(* PLC project Система умного дома.project, CODESYS CODESYS V3.5 SP17 Patch 3 *)
(* stored: creationDateTime 2026-04-06T20:38:17.5908527, modificationDateTime 2026-03-25T09:46:39.3897592 *)

TYPE E_ALERT_PRIORITY : (ALERT_PRIORITY_NONE := 0, ALERT_PRIORITY_LOW := 1, ALERT_PRIORITY_MEDIUM := 2, ALERT_PRIORITY_HIGH := 3, ALERT_PRIORITY_CRITICAL := 4) USINT;
END_TYPE

TYPE E_Adapt_Profile : (ADAPT_PROFILE_STABLE := 0, ADAPT_PROFILE_BALANCED := 1, ADAPT_PROFILE_AGGRESSIVE := 2) USINT;
END_TYPE

TYPE E_Behavior_Mode : (BEHAVIOR_HOME := 0, BEHAVIOR_AWAY := 1, BEHAVIOR_NIGHT := 2, BEHAVIOR_MAINTENANCE := 3) INT;
END_TYPE

TYPE E_FABRIC_LIFECYCLE_STATE : (FABRIC_INITIALIZING := 0, FABRIC_ACTIVE := 1, FABRIC_DEGRADED := 2, FABRIC_PASSIVE := 3, FABRIC_QUARANTINED := 4, FABRIC_SUSPENDED := 5) INT;
END_TYPE

TYPE E_GOVERNANCE_PRIORITY_TIER : (TIER_0_SAFETY := 0, TIER_1_AUTHORITY := 1, TIER_2_PHYSICAL_TRUTH := 2, TIER_3_SURVIVABILITY := 3, TIER_4_OBSERVABILITY := 4, TIER_5_ANALYTICS := 5) INT;
END_TYPE

TYPE E_Gateway_Command_Type : (CMD_NONE := 0, CMD_SET_SCENARIO := 1, CMD_SET_LIGHT := 2, CMD_SET_SOCKET := 3, CMD_SET_SECURITY := 4, CMD_SET_TEMP := 5, CMD_SET_VENT := 6, CMD_SET_BLINDS := 7, CMD_TELEGRAM_MSG := 8, CMD_SYNC_TIME := 9, CMD_RESET_ERRORS := 10, CMD_SET_CONFIG := 11) USINT;
END_TYPE

TYPE E_Heating_Allocation_Block_Reason : (NONE := 0, PRESSURE_UNAVAILABLE := 1, SERVICE_DISABLED := 2, PREDICTIVE_DEGRADED := 3, POLICY_BUDGET_SHED := 4, FREEZE_BYPASS := 5, DHW_BYPASS := 6) INT;
END_TYPE

TYPE E_Heating_Policy_Mode : (HPM_NORMAL := 0, HPM_DEGRADED := 1, HPM_FREEZE_PROTECT := 2, HPM_MAINTENANCE := 3, HPM_SAFETY_BLOCK := 4, HPM_FAULT_ISOLATION := 5) INT;
END_TYPE

TYPE E_Heating_RootCause : (RC_NONE := 0, RC_EMERGENCY_STOP := 1, RC_GAS_SAFETY := 2, RC_IO_OFFLINE := 3, RC_BOILER_OFFLINE := 4, RC_BOILER_ERROR := 5, RC_NO_FLAME := 6, RC_NO_FLOW := 7, RC_PUMP_FAILURE := 8, RC_VALVES_CLOSED := 9, RC_NO_HEAT_TRANSFER := 10, RC_LOW_SUPPLY_TEMP := 11, RC_SENSOR_ERROR := 12, RC_POLICY_BLOCKED := 13, RC_UNKNOWN := 14) INT;
END_TYPE

TYPE E_Heating_Runtime_Phase : (HRP_DISABLED := 0, HRP_IDLE := 10, HRP_DHW := 20, HRP_HEATING := 30, HRP_SERVICE_GATING := 40, HRP_STATE_PUBLICATION := 50, HRP_DIAGNOSTICS := 60, HRP_OUTPUT_PROJECTION := 70, HRP_COMPLETE := 100, HRP_FAULT := 900) INT;
END_TYPE

TYPE E_Lifetime_Device_Type : (LIFETIME_DEVICE_PUMP := 1, LIFETIME_DEVICE_FAN := 2) USINT;
END_TYPE

TYPE E_Modbus_Function : (MB_NONE := 0, MB_FC03_READ_HOLDING_REGISTERS := 3, MB_FC04_READ_INPUT_REGISTERS := 4, MB_FC06_WRITE_SINGLE_REGISTER := 6, MB_FC16_WRITE_MULTIPLE_REGISTERS := 16) INT;
END_TYPE

TYPE E_Modbus_RTU_RX_State : (MB_RTU_RX_IDLE := 0, MB_RTU_RX_RECEIVING := 1, MB_RTU_RX_FRAME_READY := 2, MB_RTU_RX_CRC_ERROR := 3, MB_RTU_RX_OVERFLOW := 4, MB_RTU_RX_SHORT_FRAME := 5) INT;
END_TYPE

TYPE E_Modbus_SysCom_Backend_State : (MB_SYSCOM_CLOSED := 0, MB_SYSCOM_OPENING := 1, MB_SYSCOM_ONLINE := 2, MB_SYSCOM_ERROR := 3, MB_SYSCOM_RECONNECT_WAIT := 4) INT;
END_TYPE

TYPE E_OpenTherm_Adapter_State : (OT_STATE_OFFLINE := 0, OT_STATE_ONLINE := 1, OT_STATE_HEARTBEAT_TIMEOUT := 2, OT_STATE_ACK_TIMEOUT := 3, OT_STATE_ADAPTER_ERROR := 4) INT;
END_TYPE

TYPE E_OpenTherm_Error : (OT_ERROR_NONE := 0, OT_ERROR_HEARTBEAT_TIMEOUT := 1, OT_ERROR_ACK_TIMEOUT := 2, OT_ERROR_ADAPTER_FAULT := 3, OT_ERROR_COMMUNICATION := 4, OT_ERROR_INVALID_RESPONSE := 5) INT;
END_TYPE

TYPE E_Outdoor_Mode : (OUTDOOR_MODE_AUTO := 0, OUTDOOR_MODE_PARTY := 1, OUTDOOR_MODE_SECURITY := 2, OUTDOOR_MODE_ECONOMY := 3, OUTDOOR_MODE_MANUAL := 4) USINT;
END_TYPE

TYPE E_PLC_ROLE : (ROLE_UNDEFINED := 0, ROLE_ACTIVE := 1, ROLE_STANDBY := 2, ROLE_OFFLINE := 3) USINT;
END_TYPE

TYPE E_RUNTIME_ADAPTIVE_MODE : (FULL_SEMANTIC_MODE := 0, REDUCED_ANALYTICS_MODE := 1, SURVIVABILITY_MODE := 2, MINIMAL_SAFE_MODE := 3) INT;
END_TYPE

TYPE E_RUNTIME_TRANSITION_RESULT : (TRANSITION_VALID := 0, TRANSITION_FORBIDDEN := 1, TRANSITION_REQUIRES_PROOF := 2, TRANSITION_REQUIRES_RECOVERY := 3, TRANSITION_REQUIRES_TEMPORAL_ALIGNMENT := 4) INT;
END_TYPE

TYPE E_Recovery_Phase : (IDLE := 0, STABILIZING := 1, WAIT_MANUAL_CONFIRM := 2, RECOVERING := 3, COOLDOWN := 4, ABORTED := 5) USINT;
END_TYPE

TYPE E_Rule_Action_Type : (ACTION_NONE := 0, ACTION_SET_FLOOR_HEATING := 1, ACTION_SET_LIGHTING_BASE := 2, ACTION_SET_LIGHTING_ACCENT := 3, ACTION_SET_SOCKET := 4, ACTION_SET_VENTILATION := 5, ACTION_SET_BLINDS := 6, ACTION_ACTIVATE_SCENARIO := 7, ACTION_TOGGLE_LIGHTING := 8, ACTION_TOGGLE_SOCKET := 9) USINT;
END_TYPE

TYPE E_Rule_Comparison : (COMP_NONE := 0, COMP_EQ := 1, COMP_GT := 2, COMP_LT := 3, COMP_GE := 4, COMP_LE := 5, COMP_IN_RANGE := 6, COMP_TRUE := 7, COMP_FALSE := 8) USINT;
END_TYPE

TYPE E_Rule_Condition_Type : (COND_NONE := 0, COND_AIR_TEMP := 1, COND_FLOOR_TEMP := 2, COND_HUMIDITY := 3, COND_CO2 := 4, COND_METHANE := 5, COND_CO := 6, COND_DOOR_WINDOW := 7, COND_FLOOD := 8, COND_SMOKE := 9, COND_MOTION := 10, COND_TIME_OF_DAY := 11, COND_DAY_OF_WEEK := 12) USINT;
END_TYPE

TYPE E_Runtime_Observer_Lifecycle_State : (ROS_INACTIVE := 0, ROS_AUTHORIZATION_PENDING := 10, ROS_AUTHORIZATION_DENIED := 20, ROS_STABILIZATION := 30, ROS_OPERATIONAL := 40, ROS_ROLLBACK := 50, ROS_FAULTED := 900) INT;
END_TYPE

TYPE E_SCENARIO_SOURCE : (SRC_NONE := 0, SRC_OPERATOR := 1, SRC_GATEWAY := 2, SRC_RULE := 3, SRC_SAFETY := 4, SRC_POLICY := 5) INT;
END_TYPE

TYPE E_SCENARIO_TYPE : (SCENARIO_NONE := 0, SCENARIO_MORNING := 1, SCENARIO_EVENING := 2, SCENARIO_AWAY := 3, SCENARIO_PARTY := 4, SCENARIO_SLEEP := 5, SCENARIO_EMERGENCY := 6, SCENARIO_PRESENCE := 7) USINT;
END_TYPE

TYPE E_SEMANTIC_EXECUTION_PATH : (FAST_PATH := 0, NORMAL_PATH := 1, DEFERRED_PATH := 2, BACKGROUND_PATH := 3) INT;
END_TYPE

TYPE E_SENSOR_TYPE : (SENSOR_TYPE_NONE := 0, SENSOR_TYPE_DOOR_WINDOW := 5, SENSOR_TYPE_GLASS_BREAK := 6, SENSOR_TYPE_FLOOD := 7, SENSOR_TYPE_SMOKE := 8, SENSOR_TYPE_GAS_METHANE := 1, SENSOR_TYPE_GAS_CO := 2, SENSOR_TYPE_TEMP_FLOOR := 3, SENSOR_TYPE_TEMP_AIR := 4, SENSOR_TYPE_CO2 := 9) USINT;
END_TYPE

TYPE E_SYSTEM_RUNTIME_STATE : (SYS_SAFE := 0, SYS_DEGRADED := 1, SYS_RECOVERING := 2, SYS_QUARANTINED := 3, SYS_ISOLATED := 4, SYS_PARTITIONED := 5, SYS_TRUSTLESS := 6) INT;
END_TYPE

TYPE E_Safety_Mode : (NORMAL := 0, FIRE := 1, GAS := 2, WATER_LEAK := 3, GLOBAL_STOP := 4) USINT;
END_TYPE

TYPE E_System_Operating_Mode : (MODE_NORMAL := 0, MODE_DEGRADED := 1, MODE_SAFE_STOP := 2, MODE_FREEZE_PROTECTION := 3) INT;
END_TYPE

TYPE E_System_Reason_Code : (REASON_NONE := 0, REASON_USER := 1, REASON_SAFETY := 2, REASON_AUTOMATION := 3, REASON_INTERNAL := 4, REASON_SCENARIO_VENT_BOOST := 5, REASON_USER_REQUEST := 6, REASON_SCENARIO_NIGHT := 7, REASON_DOMAIN_PROJECTION := 8, REASON_SAFETY_BLOCK := 9) USINT;
END_TYPE

TYPE E_System_Root_Cause : (ROOT_NONE := 0, ROOT_FIRE := 1, ROOT_GAS_LEAK := 2, ROOT_CO_WARNING := 3, ROOT_CO_CRITICAL := 4, ROOT_WATER_LEAK := 5, ROOT_IO_OFFLINE := 6, ROOT_COMM_FAULT := 7, ROOT_SENSOR_FAULT := 8, ROOT_SUBSYSTEM_FAULT := 9, ROOT_WATCHDOG_FAULT := 10) INT;
END_TYPE

TYPE E_System_Severity : (SEV_NORMAL := 0, SEV_WARNING := 1, SEV_DEGRADED := 2, SEV_CRITICAL := 3) INT;
END_TYPE

TYPE E_Trace_Layer : (TRACE_SYSTEM := 0, TRACE_SAFETY := 1, TRACE_HEATING := 2, TRACE_IO := 3, TRACE_SCENARIO := 4, TRACE_USER := 5) USINT;
END_TYPE

TYPE E_Trace_Source : (SRC_MAIN := 0, SRC_IO := 1, SRC_DIAGNOSTICS := 2, SRC_HEATING := 3, SRC_SCENARIO := 4, SRC_USER := 5) USINT;
END_TYPE

TYPE E_Trend_Parameter_Type : (TREND_PARAM_NONE := 0, TREND_PARAM_TEMP_AIR := 1, TREND_PARAM_TEMP_FLOOR := 2, TREND_PARAM_PRESSURE := 3, TREND_PARAM_PUMP_CURRENT := 4, TREND_PARAM_GAS_METHANE := 5, TREND_PARAM_GAS_CO := 6) USINT;
END_TYPE

TYPE E_TwoFactor_Method : (TF_METHOD_NONE := 0, TF_METHOD_RFID := 1, TF_METHOD_TOTP := 2, TF_METHOD_BOTH := 3) USINT;
END_TYPE

TYPE E_VALVE_TYPE : (VALVE_NC := 1, VALVE_NO := 2) USINT;
END_TYPE

TYPE E_VENTILATION_LOCATION : (VENT_LOCATION_NONE := 0, VENT_LOCATION_BASEMENT_GAME_ROOM := 1, VENT_LOCATION_BASEMENT_GYM := 2, VENT_LOCATION_BASEMENT_BOILER_ROOM := 3, VENT_LOCATION_BATHROOM_1F := 4, VENT_LOCATION_BATHROOM_2F := 5, VENT_LOCATION_MASTER_BATHROOM := 6, VENT_LOCATION_LAUNDRY := 7, VENT_LOCATION_KITCHEN := 8) USINT;
END_TYPE

TYPE E_VENTILATION_UNIT_TYPE : (VENTILATION_TYPE_NONE := 0, VENTILATION_TYPE_SUPPLY := 1, VENTILATION_TYPE_EXHAUST := 2) USINT;
END_TYPE

TYPE E_Valve_Test_Result : (TEST_RESULT_NONE := 0, TEST_RESULT_PASSED := 1, TEST_RESULT_CURRENT_DEVIATION := 2, TEST_RESULT_TIME_DEVIATION := 3, TEST_RESULT_STALL := 4, TEST_RESULT_LIMIT_SWITCH_FAIL := 5, TEST_RESULT_ABORTED := 6) USINT;
END_TYPE

TYPE E_WEATHER_COMPENSATION_METHOD : (WEATHER_COMP_NONE := 0, WEATHER_COMP_OUTDOOR_RESET := 1) USINT;
END_TYPE

TYPE E_Zone_Access_Level : (ZONE_ACCESS_NONE := 0, ZONE_ACCESS_VIEW := 1, ZONE_ACCESS_CONTROL := 2, ZONE_ACCESS_CONFIG := 3, ZONE_ACCESS_FULL := 4) USINT;
END_TYPE

TYPE ST_Alarm_Record : STRUCT
  ID : UDINT;
  Timestamp_MS : UDINT;
  Source : STRING(20);
  Source_ID : BYTE;
  Message : STRING(100);
  Severity : E_ALERT_PRIORITY;
  Is_Active : BOOL;
  Is_Acknowledged : BOOL;
END_STRUCT;
END_TYPE

TYPE ST_Astro_Time : STRUCT
  sunrise_ms : UDINT := 0;
  sunset_ms : UDINT := 0;
  is_daylight : BOOL := FALSE;
END_STRUCT;
END_TYPE

TYPE ST_Behavior_Weights : STRUCT
  W_Comfort : REAL;
  W_Night : REAL;
  W_Preheat : REAL;
  W_VentBoost : REAL;
  W_AccessSecure : REAL;
END_STRUCT;
END_TYPE

TYPE ST_BlackBox_Record : STRUCT
  Timestamp : UDINT;
  Gas_Methane_LEL : REAL;
  Gas_CO_PPM : REAL;
  Flood_Active : BOOL;
  Fire_Active : BOOL;
  Valve_Gas_Status : BYTE;
  Valve_Water_Status : BYTE;
  PLC_Active_ID : BYTE;
  System_Mode : BYTE;
  First_Fault_Type : BYTE;
  First_Fault_Source : BYTE;
  First_Fault_Active : BOOL;
  System_Severity : BYTE;
  Root_Cause : BYTE;
  Watchdog_Fault : BOOL;
END_STRUCT;
END_TYPE

TYPE ST_Boiler_Status : STRUCT
  Active : BOOL;
  Running : BOOL;
  Warning : BOOL;
  Error : BOOL;
  Error_ID : WORD;
  Power_Percent : REAL;
  Current_Power : REAL;
  Work_Seconds : UDINT;
  Work_Hours : REAL;
  Resource_Percent : REAL := 100.0;
  Last_Start : DT;
  OT_Online : BOOL;
  OT_Command_Valid : BOOL;
  OT_Transport_Degraded : BOOL;
  OT_Adapter_Error : BOOL;
  Available : BOOL;
  Selected_By_Cascade : BOOL;
  Flame_Missing : BOOL;
  Transport_Missing : BOOL;
  Ignition_Timeout : BOOL;
  Degraded : BOOL;
END_STRUCT;
END_TYPE

TYPE ST_Calibration_Family_Summary : STRUCT
  active : BOOL;
  status : INT;
  sensor_count : INT;
  verification_active_count : INT;
  failed_count : INT;
  max_deviation_percent : REAL;
  summary_text : STRING(160);
END_STRUCT;
END_TYPE

TYPE ST_Calibration_Sensor_Summary : STRUCT
  active : BOOL;
  status : INT;
  calibrated_value : REAL;
  deviation_percent : REAL;
  verification_active : BOOL;
  verification_failed : BOOL;
  record_index : INT;
  label : STRING(64);
  summary_text : STRING(160);
END_STRUCT;
END_TYPE

TYPE ST_Component_Maintenance : STRUCT
  Is_Faulty : BOOL;
  Is_In_Maintenance : BOOL;
  Fallback_Value : REAL;
  Use_Last_Good_Value : BOOL;
END_STRUCT;
END_TYPE

TYPE ST_Config_Activation_State : STRUCT
  Runtime_Valid : BOOL;
  Runtime_System_Time_MS : UDINT;
  Active_Version : UDINT;
  Staged_Version : UDINT;
  Previous_Stable_Version : UDINT;
  Staged_Config_Valid : BOOL;
  Activation_Requested : BOOL;
  Activation_Allowed : BOOL;
  Activation_Blocked : BOOL;
  Rollback_Requested : BOOL;
  Rollback_Available : BOOL;
  Rollback_Active : BOOL;
  Config_Quarantine_Active : BOOL;
  Migration_Required : BOOL;
  Migration_Compatible : BOOL;
  Status_Code : UINT;
  Status_Text : STRING(160);
END_STRUCT;
END_TYPE

TYPE ST_DHW_Config : STRUCT
  Target_Temp : REAL := 55.0;
  Hysteresis : REAL := 2.0;
  Circulation_Schedule_Enabled : BOOL := TRUE;
  Circulation_Start : TOD := TOD#06:00;
  Circulation_End : TOD := TOD#23:00;
  Night_Mode_Enabled : BOOL := TRUE;
  Anti_Legionella_Enabled : BOOL := TRUE;
  Anti_Legionella_Day : UINT := 7;
  Degraded_Target_Delta : REAL := 5.0;
END_STRUCT;
END_TYPE

TYPE ST_DHW_Status : STRUCT
  Temp : REAL;
  Pressure : REAL;
  Heating_Pump_On : BOOL;
  Circ_Pump_On : BOOL;
  Warning : BOOL;
  Error : BOOL;
  Error_ID : WORD;
END_STRUCT;
END_TYPE

TYPE ST_Device_Health : STRUCT
  Health_Score : BYTE := 100;
  Total_Runtime_Hours : UDINT;
  Starts_Count : UDINT;
  Last_Start_Current : REAL;
  Avg_Start_Current : REAL;
  Sample_Count : UDINT;
  Current_Sum : REAL;
  Maintenance_Required : BOOL;
  Warning_Message : STRING(50);
END_STRUCT;
END_TYPE

TYPE ST_Diagnostic_Event : STRUCT
  Code : UDINT;
  Severity : INT;
  Active : BOOL;
  Timestamp : UDINT;
  Source : INT;
END_STRUCT;
END_TYPE

TYPE ST_Distributed_Authority_State : STRUCT
  Runtime_Valid : BOOL;
  Runtime_System_Time_MS : UDINT;
  Controller_Id : UINT;
  Runtime_Node_Id : UINT;
  Authority_Domain_Id : UINT;
  Authority_Election_Active : BOOL;
  Authority_Master_Elected : BOOL;
  Authority_Backup_Elected : BOOL;
  Authority_Observer_Only : BOOL;
  Authority_Lease_Valid : BOOL;
  Authority_Lease_Expired : BOOL;
  Authority_Lease_Timeout_MS : UDINT;
  Replication_Consensus_Healthy : BOOL;
  Replication_Consensus_Stale : BOOL;
  Recovery_Authority_Allowed : BOOL;
  Rollback_Authority_Allowed : BOOL;
  Quarantine_Authority_Allowed : BOOL;
  Split_Brain_Blocked : BOOL;
  Distributed_Safety_Barrier_OK : BOOL;
  Status_Code : UINT;
  Status_Text : STRING(160);
END_STRUCT;
END_TYPE

TYPE ST_Distributed_Orchestration_State : STRUCT
  Runtime_Valid : BOOL;
  Runtime_System_Time_MS : UDINT;
  Orchestration_Sequence_Id : UDINT;
  Distributed_Execution_Active : BOOL;
  Cross_Node_Isolation_Required : BOOL;
  Cross_Node_Recovery_Required : BOOL;
  Cross_Node_Rollback_Required : BOOL;
  Distributed_Projection_Granted : BOOL;
  Distributed_Projection_Blocked : BOOL;
  Distributed_Rollback_Allowed : BOOL;
  Distributed_Recovery_Allowed : BOOL;
  Distributed_Scheduler_Healthy : BOOL;
  Distributed_Timing_Window_Valid : BOOL;
  Remote_Node_Ack_Required : BOOL;
  Remote_Node_Ack_Received : BOOL;
  Distributed_Conflict_Detected : BOOL;
  Distributed_Split_Execution_Suspected : BOOL;
  Status_Code : UINT;
  Status_Text : STRING(160);
END_STRUCT;
END_TYPE

TYPE ST_Distributed_Projection_Ownership : STRUCT
  Ownership_Valid : BOOL;
  Runtime_System_Time_MS : UDINT;
  Projection_Id : UINT;
  Projection_Class : UINT;
  Owner_Controller_Id : UINT;
  Owner_Runtime_Node_Id : UINT;
  Owner_Authority_Domain_Id : UINT;
  Ownership_Granted : BOOL;
  Ownership_Revoked : BOOL;
  Ownership_Conflict : BOOL;
  Ownership_Stale : BOOL;
  Projection_Active : BOOL;
  Projection_Blocked : BOOL;
  Distributed_Execution_Allowed : BOOL;
  Distributed_Recovery_Allowed : BOOL;
  Status_Code : UINT;
  Status_Text : STRING(160);
END_STRUCT;
END_TYPE

TYPE ST_Distributed_Recovery_Lock : STRUCT
  Lock_Valid : BOOL;
  Runtime_System_Time_MS : UDINT;
  Lock_Id : UDINT;
  Lock_Sequence_Id : UDINT;
  Owner_Controller_Id : UINT;
  Owner_Runtime_Node_Id : UINT;
  Recovery_Lock_Active : BOOL;
  Rollback_Lock_Active : BOOL;
  Reopen_Lock_Active : BOOL;
  Lock_Conflict : BOOL;
  Lock_Expired : BOOL;
  Lock_Revoked : BOOL;
  Distributed_Execution_Allowed : BOOL;
  Status_Code : UINT;
  Status_Text : STRING(160);
END_STRUCT;
END_TYPE

TYPE ST_Distributed_Runtime_Message : STRUCT
  Message_Valid : BOOL;
  Message_Time_MS : UDINT;
  Message_Id : UDINT;
  Source_Controller_Id : UINT;
  Source_Runtime_Node_Id : UINT;
  Target_Runtime_Node_Id : UINT;
  Message_Class : UINT;
  Message_Version : UINT;
  Authority_State_Replicated : BOOL;
  Recovery_State_Replicated : BOOL;
  Quarantine_State_Replicated : BOOL;
  Topology_State_Replicated : BOOL;
  Binding_State_Replicated : BOOL;
  Replication_Sequence_Id : UDINT;
  Replication_Ack_Required : BOOL;
  Replication_Ack_Received : BOOL;
  Status_Code : UINT;
  Status_Text : STRING(160);
END_STRUCT;
END_TYPE

TYPE ST_Distributed_Runtime_Node_State : STRUCT
  Runtime_Valid : BOOL;
  Runtime_System_Time_MS : UDINT;
  Controller_Id : UINT;
  Runtime_Node_Id : UINT;
  Authority_Domain_Id : UINT;
  Topology_Domain_Id : UINT;
  Node_Online : BOOL;
  Node_Degraded : BOOL;
  Node_Quarantined : BOOL;
  Node_Backup_Mode : BOOL;
  Node_Observer_Mode : BOOL;
  Authority_Allowed : BOOL;
  Authority_Revoked : BOOL;
  Authority_Master : BOOL;
  Authority_Backup : BOOL;
  Replication_Healthy : BOOL;
  Replication_Timeout : BOOL;
  Split_Brain_Suspected : BOOL;
  Restart_Continuity_Valid : BOOL;
  Quarantine_State_Replicated : BOOL;
  Recovery_State_Replicated : BOOL;
  Status_Code : UINT;
  Status_Text : STRING(160);
END_STRUCT;
END_TYPE

TYPE ST_Distributed_Topology_Domain : STRUCT
  Domain_Valid : BOOL;
  Domain_Id : UINT;
  Controller_Id : UINT;
  Runtime_Node_Id : UINT;
  Authority_Owner : BOOL;
  Backup_Owner : BOOL;
  Observer_Only : BOOL;
  Domain_Online : BOOL;
  Domain_Degraded : BOOL;
  Domain_Quarantined : BOOL;
  Cross_Node_Dependencies : BOOL;
  Remote_Valve_Group_Required : BOOL;
  Remote_Recovery_Required : BOOL;
  Distributed_Path_Valid : BOOL;
  Distributed_Projection_Allowed : BOOL;
  Status_Code : UINT;
  Status_Text : STRING(160);
END_STRUCT;
END_TYPE

TYPE ST_EVENT : STRUCT
  Event_ID : UDINT;
  Event_Type : UINT;
  Timestamp : UDINT;
  Param1 : UDINT;
  Param2 : UDINT;
END_STRUCT;
END_TYPE

TYPE ST_Flood_Config : STRUCT
  Emergency_Two_Stage_Enabled : BOOL := TRUE;
  Valve_Test_Period_Days : UINT := 7;
  Current_Threshold_MA : REAL := 500.0;
  sensor_to_valve_map : ARRAY[1..GVL_CONSTANTS.C_MAX_FLOOD_SENSORS] OF INT := [1, 1, 1, 1, 2, 2, 2, 2, 3, 3, 3, 3];
END_STRUCT;
END_TYPE

TYPE ST_Flood_Global_Config : STRUCT
  valve_types : ARRAY[1..GVL_CONSTANTS.C_MAX_FLOOD_VALVES] OF E_VALVE_TYPE := [GVL_CONSTANTS.C_MAX_FLOOD_VALVES(E_VALVE_TYPE.VALVE_NC)];
  sensor_to_valve_map : ARRAY[1..GVL_CONSTANTS.C_MAX_FLOOD_SENSORS] OF BYTE := [1, 1, 1, 2, 2, 2, 2, 0, 0, 0];
  min_duration_ms : UDINT := 5000;
  warning_duration_ms : UDINT := 30000;
END_STRUCT;
END_TYPE

TYPE ST_FloorHeating_Circuit_Config : STRUCT
  circuit_id : BYTE := 0;
  zone : BYTE := 0;
  manifold_id : BYTE := 1;
  sensor_id : BYTE := 1;
  valve_id : BYTE := 1;
  control_type : BYTE := 1;
  design_temp : REAL := 35.0;
  min_temp : REAL := 20.0;
  max_temp : REAL := 45.0;
  pid_kp : REAL := 2.0;
  pwm_period_s : UINT := 600;
END_STRUCT;
END_TYPE

TYPE ST_FloorHeating_Global_Config : STRUCT
  enable_floor_heating : BOOL := TRUE;
  anti_freeze_temp : REAL := 7.0;
  overheat_temp : REAL := 45.0;
  weather_compensation_enabled : BOOL := TRUE;
  total_circuits : BYTE := 16;
END_STRUCT;
END_TYPE

TYPE ST_FloorHeating_Manifold_Config : STRUCT
  manifold_id : BYTE;
  location : STRING(30);
  nominal_flow : REAL;
  enable_pump : BOOL;
  circuits : ARRAY[1..GVL_CONSTANTS.C_MAX_CIRCUITS_PER_MANIFOLD] OF ST_FloorHeating_Circuit_Config;
END_STRUCT;
END_TYPE

TYPE ST_Forensic_Journal_Record : STRUCT
  Record_Valid : BOOL;
  Event_Time_MS : UDINT;
  Event_Id : UDINT;
  Event_Class : UINT;
  Event_Severity : UINT;
  Config_Version : UDINT;
  Topology_Version : UDINT;
  Recovery_Domain_Id : UINT;
  Valve_Group_Id : UINT;
  Sensor_Id : UINT;
  Activation_Event : BOOL;
  Rollback_Event : BOOL;
  Quarantine_Event : BOOL;
  Recovery_Event : BOOL;
  Restart_Event : BOOL;
  Status_Code : UINT;
  Event_Text : STRING(160);
END_STRUCT;
END_TYPE

TYPE ST_Gas_Valve_Configuration : STRUCT
  valve_id : BYTE := 0;
  valve_type : E_VALVE_TYPE := E_VALVE_TYPE.VALVE_NC;
  close_time_seconds : UDINT := 10;
  open_time_seconds : UDINT := 10;
  emergency_open_allowed : BOOL := FALSE;
END_STRUCT;
END_TYPE

TYPE ST_Gateway_Command : STRUCT
  command_id : UDINT;
  timestamp_ms : UDINT;
  operator_id : STRING(10);
  command_type : E_Gateway_Command_Type;
  target_zone : BYTE;
  target_value : REAL;
  target_on_off : BOOL;
  target_scenario : E_SCENARIO_TYPE;
  target_armed : BOOL;
  target_pin : STRING(4);
  target_2fa_code : STRING(6);
  telegram_msg : STRING(200);
  source_ip : STRING(15);
  crc32 : DWORD;
END_STRUCT;
END_TYPE

TYPE ST_HMI_Config_Workflow_State : STRUCT
  Runtime_Valid : BOOL;
  Runtime_System_Time_MS : UDINT;
  Editor_Open : BOOL;
  Edit_Session_Active : BOOL;
  Draft_Dirty : BOOL;
  Validation_Requested : BOOL;
  Validation_OK : BOOL;
  Validation_Failed : BOOL;
  Activation_Requested : BOOL;
  Activation_Allowed : BOOL;
  Activation_Blocked : BOOL;
  Rollback_Requested : BOOL;
  Rollback_Allowed : BOOL;
  Operator_Ack_Required : BOOL;
  Service_Mode_Required : BOOL;
  Quarantine_Visible : BOOL;
  Active_Version : UDINT;
  Draft_Version : UDINT;
  Last_Stable_Version : UDINT;
  Status_Code : UINT;
  Status_Text : STRING(160);
END_STRUCT;
END_TYPE

TYPE ST_Heating_Circuit_Runtime_Projection : STRUCT
  Visible : BOOL;
  Selected_Source_Code : UINT;
  Selected_Source_Confidence : REAL;
  Fallback_Active : BOOL;
  Source_Degraded : BOOL;
  Sensor_Error_Active : BOOL;
  Reason_Code : UINT;
  Reason_Text : STRING(128);
  Source_Switched_Event : BOOL;
  Fallback_Activated_Event : BOOL;
  Fallback_Recovered_Event : BOOL;
  Source_Loss_Event : BOOL;
  Last_Event_Code : UINT;
  Last_Event_Text : STRING(128);
  Last_Event_MS : UDINT;
END_STRUCT;
END_TYPE

TYPE ST_Heating_Config : STRUCT
  Weather_Comp_Enabled : BOOL := TRUE;
  Weather_Coef : REAL := 0.1;
  Freeze_Threshold : REAL := 7.0;
  Overheat_Threshold : REAL := 45.0;
  Night_Reduction : REAL := 3.0;
  Target_Floor_Temp : REAL := 28.0;
  Target_Room_Temp : REAL := 22.0;
  Hysteresis : REAL := 0.5;
END_STRUCT;
END_TYPE

TYPE ST_Heating_Runtime_Adaptive_Intelligence : STRUCT
  Adaptive_Analytics_Visible : BOOL;
  Adaptive_Analytics_Degraded : BOOL;
  Adaptive_Analytics_Attention : BOOL;
  Supervision_Confidence_Observation : UINT;
  Confidence_Degradation_Visible : BOOL;
  Adaptive_Runtime_Observation : UINT;
  Adaptive_Runtime_Stability_Observation : UINT;
  Runtime_Anomaly_Observation_Weight : UINT;
  Cascade_Anomaly_Observation_Weight : UINT;
  OpenTherm_Anomaly_Observation_Weight : UINT;
  Diagnostics_Anomaly_Observation_Weight : UINT;
  Predictive_Correlation_Observation : UINT;
  Predictive_Correlation_Visible : BOOL;
  Sequencing_Confidence_Observation : UINT;
  Ownership_Confidence_Observation : UINT;
  Synchronization_Confidence_Observation : UINT;
  Status_Code : UINT;
  Status_Text : STRING(128);
END_STRUCT;
END_TYPE

TYPE ST_Heating_Runtime_Anomaly : STRUCT
  Anomaly_Active : BOOL;
  Anomaly_Acknowledged : BOOL;
  Anomaly_Cleared : BOOL;
  Runtime_Jitter_Detected : BOOL;
  Runtime_Latency_Detected : BOOL;
  Runtime_Degraded : BOOL;
  Cascade_Degraded : BOOL;
  Cascade_Boiler_Loss_Detected : BOOL;
  OpenTherm_Transport_Degraded : BOOL;
  OpenTherm_Command_Invalid : BOOL;
  Diagnostics_Degraded : BOOL;
  Explainability_Degraded : BOOL;
  Sequencing_Invalid : BOOL;
  Ownership_Invalid : BOOL;
  Synchronization_Invalid : BOOL;
  Severity_Level : UINT;
  Critical_Anomaly : BOOL;
  Status_Code : UINT;
  Status_Text : STRING(128);
END_STRUCT;
END_TYPE

TYPE ST_Heating_Runtime_Blackbox_Event : STRUCT
  Event_ID : UDINT;
  Event_Active : BOOL;
  Runtime_Phase : E_Heating_Runtime_Phase;
  Event_Start_MS : UDINT;
  Event_End_MS : UDINT;
  Event_Duration_MS : UDINT;
  Runtime_Degraded : BOOL;
  Runtime_Fault : BOOL;
  Cascade_Degraded : BOOL;
  Cascade_Boiler_Loss : BOOL;
  OpenTherm_Degraded : BOOL;
  OpenTherm_Command_Invalid : BOOL;
  Sequencing_Invalid : BOOL;
  Ownership_Invalid : BOOL;
  Synchronization_Invalid : BOOL;
  Root_Cause_Candidate : BOOL;
  Critical_Path : BOOL;
  Status_Code : UINT;
  Status_Text : STRING(128);
END_STRUCT;
END_TYPE

TYPE ST_Heating_Runtime_Blackbox_Timeline : STRUCT
  Events : ARRAY[1..256] OF ST_Heating_Runtime_Blackbox_Event;
  Write_Index : UINT;
  Event_Count : UINT;
  Timeline_Overflow : BOOL;
  Reconstruction_Visible : BOOL;
  Forensic_Timeline_Visible : BOOL;
  Root_Cause_Reconstructed : BOOL;
  Sequencing_Valid : BOOL;
  Ownership_Valid : BOOL;
  Synchronization_Valid : BOOL;
  Status_Code : UINT;
  Status_Text : STRING(128);
END_STRUCT;
END_TYPE

TYPE ST_Heating_Runtime_Causality_Edge : STRUCT
  Source_Node_ID : UINT;
  Target_Node_ID : UINT;
  Edge_Active : BOOL;
  Propagation_Detected : BOOL;
  Runtime_Propagation : BOOL;
  Cascade_Propagation : BOOL;
  OpenTherm_Propagation : BOOL;
  Diagnostics_Propagation : BOOL;
  Sequencing_Propagation : BOOL;
  Ownership_Propagation : BOOL;
  Synchronization_Propagation : BOOL;
  Severity_Level : UINT;
  Critical_Path : BOOL;
  Status_Code : UINT;
  Status_Text : STRING(128);
END_STRUCT;
END_TYPE

TYPE ST_Heating_Runtime_Causality_Graph : STRUCT
  Nodes : ARRAY[1..64] OF ST_Heating_Runtime_Causality_Node;
  Edges : ARRAY[1..128] OF ST_Heating_Runtime_Causality_Edge;
  Node_Count : UINT;
  Edge_Count : UINT;
  Graph_Active : BOOL;
  Graph_Degraded : BOOL;
  Graph_Critical : BOOL;
  Sequencing_Valid : BOOL;
  Ownership_Valid : BOOL;
  Synchronization_Valid : BOOL;
  Status_Code : UINT;
  Status_Text : STRING(128);
END_STRUCT;
END_TYPE

TYPE ST_Heating_Runtime_Causality_Node : STRUCT
  Node_ID : UINT;
  Node_Active : BOOL;
  Runtime_Degraded : BOOL;
  Runtime_Fault : BOOL;
  Cascade_Degraded : BOOL;
  Cascade_Boiler_Loss : BOOL;
  OpenTherm_Degraded : BOOL;
  OpenTherm_Command_Invalid : BOOL;
  Diagnostics_Degraded : BOOL;
  Explainability_Degraded : BOOL;
  Sequencing_Invalid : BOOL;
  Ownership_Invalid : BOOL;
  Synchronization_Invalid : BOOL;
  Severity_Level : UINT;
  Root_Cause_Candidate : BOOL;
  Status_Code : UINT;
  Status_Text : STRING(128);
END_STRUCT;
END_TYPE

TYPE ST_Heating_Runtime_Context : STRUCT
  Runtime_Enabled : BOOL;
  Runtime_Ready : BOOL;
  Runtime_Fault : BOOL;
  Current_Phase : E_Heating_Runtime_Phase;
  Allow_DHW_Phase : BOOL;
  Allow_Heating_Phase : BOOL;
  Allow_Service_Gating_Phase : BOOL;
  Allow_State_Publication_Phase : BOOL;
  Allow_Diagnostics_Phase : BOOL;
  Allow_Output_Projection_Phase : BOOL;
  DHW_Executed : BOOL;
  Heating_Executed : BOOL;
  Service_Gating_Executed : BOOL;
  State_Publication_Executed : BOOL;
  Diagnostics_Executed : BOOL;
  Output_Projection_Executed : BOOL;
  DHW_Before_Heating_Valid : BOOL;
  State_Publication_Before_Diagnostics_Valid : BOOL;
  Output_Projection_Last_Valid : BOOL;
  Runtime_Status_Code : UINT;
  Runtime_Status_Text : STRING(128);
  Diagnostics_Isolation_Valid : BOOL;
  Explainability_Isolation_Valid : BOOL;
  Safety_Isolation_Valid : BOOL;
  OpenTherm_Ownership_Valid : BOOL;
  Cascade_Ownership_Valid : BOOL;
END_STRUCT;
END_TYPE

TYPE ST_Heating_Runtime_Event_Buffer : STRUCT
  Events : ARRAY[1..32] OF ST_Heating_Runtime_Phase_Event;
  Write_Index : UINT;
  Read_Index : UINT;
  Event_Count : UINT;
  Overflow : BOOL;
  Ordering_Integrity_Valid : BOOL;
  Isolation_Integrity_Valid : BOOL;
  Lifecycle_Integrity_Valid : BOOL;
  Diagnostics_Visibility_Valid : BOOL;
  Explainability_Visibility_Valid : BOOL;
  OpenTherm_Ownership_Valid : BOOL;
  Cascade_Ownership_Valid : BOOL;
  Safety_Ownership_Valid : BOOL;
  Status_Code : UINT;
  Status_Text : STRING(128);
END_STRUCT;
END_TYPE

TYPE ST_Heating_Runtime_Execution_Frame : STRUCT
  Phase : E_Heating_Runtime_Phase;
  Frame_Started : BOOL;
  Frame_Completed : BOOL;
  Frame_Failed : BOOL;
  Frame_Start_MS : UDINT;
  Frame_End_MS : UDINT;
  Frame_Duration_MS : UDINT;
  Sequencing_Valid : BOOL;
  Ownership_Valid : BOOL;
  Synchronization_Valid : BOOL;
  Runtime_Jitter_Detected : BOOL;
  Runtime_Latency_Detected : BOOL;
  Runtime_Degraded : BOOL;
  Status_Code : UINT;
  Status_Text : STRING(128);
END_STRUCT;
END_TYPE

TYPE ST_Heating_Runtime_Execution_Timeline : STRUCT
  Frames : ARRAY[1..64] OF ST_Heating_Runtime_Execution_Frame;
  Write_Index : UINT;
  Frame_Count : UINT;
  Timeline_Overflow : BOOL;
  Sequencing_Valid : BOOL;
  Ownership_Valid : BOOL;
  Synchronization_Valid : BOOL;
  Runtime_Jitter_Detected : BOOL;
  Runtime_Latency_Detected : BOOL;
  Runtime_Degraded : BOOL;
  Status_Code : UINT;
  Status_Text : STRING(128);
END_STRUCT;
END_TYPE

TYPE ST_Heating_Runtime_Integration_Bridge : STRUCT
  Shell_Ready : BOOL;
  Shell_Fault : BOOL;
  Shell_Contract_Valid : BOOL;
  Allow_DHW_Integration : BOOL;
  Allow_Heating_Integration : BOOL;
  Allow_Diagnostics_Integration : BOOL;
  Allow_Output_Projection_Integration : BOOL;
  Runtime_Ownership_Valid : BOOL;
  Diagnostics_Ownership_Valid : BOOL;
  Explainability_Ownership_Valid : BOOL;
  OpenTherm_Ownership_Valid : BOOL;
  Cascade_Ownership_Valid : BOOL;
  Safety_Ownership_Valid : BOOL;
  DHW_Before_Heating_Valid : BOOL;
  Diagnostics_After_Publication_Valid : BOOL;
  Output_Projection_Last_Valid : BOOL;
  Governance_Locked : BOOL;
  Runtime_Attachment_Allowed : BOOL;
  Runtime_Attachment_Active : BOOL;
  Integration_Status_Code : UINT;
  Integration_Status_Text : STRING(128);
  Diagnostics_Visible : BOOL;
  Explainability_Visible : BOOL;
  Current_Phase : E_Heating_Runtime_Phase;
  Runtime_Synchronized : BOOL;
END_STRUCT;
END_TYPE

TYPE ST_Heating_Runtime_Meta_Supervision : STRUCT
  Meta_Analytics_Visible : BOOL;
  Meta_Analytics_Degraded : BOOL;
  Meta_Analytics_Attention : BOOL;
  Supervision_Integrity_Visible : BOOL;
  Supervision_Integrity_Observation : UINT;
  Adaptive_Drift_Visible : BOOL;
  Adaptive_Drift_Observation : UINT;
  Confidence_Degradation_Visible : BOOL;
  Confidence_Degradation_Observation : UINT;
  Analytics_Consistency_Visible : BOOL;
  Analytics_Consistency_Observation : UINT;
  Sequencing_Meta_Observation : BOOL;
  Ownership_Meta_Observation : BOOL;
  Synchronization_Meta_Observation : BOOL;
  Status_Code : UINT;
  Status_Text : STRING(128);
END_STRUCT;
END_TYPE

TYPE ST_Heating_Runtime_Observation : STRUCT
  Runtime_Active : BOOL;
  Runtime_Ready : BOOL;
  Runtime_Fault : BOOL;
  Current_Phase : E_Heating_Runtime_Phase;
  DHW_Demand_Active : BOOL;
  DHW_Heating_Active : BOOL;
  DHW_Circulation_Active : BOOL;
  Heating_Demand_Active : BOOL;
  Heating_Runtime_Active : BOOL;
  Heating_Output_Active : BOOL;
  Cascade_Available : BOOL;
  Cascade_Degraded : BOOL;
  Cascade_Active_Boilers : UINT;
  Cascade_Available_Boilers : UINT;
  OpenTherm_Online : BOOL;
  OpenTherm_Command_Valid : BOOL;
  OpenTherm_Transport_Degraded : BOOL;
  Diagnostics_Active : BOOL;
  Explainability_Active : BOOL;
  DHW_Before_Heating_Observed : BOOL;
  Diagnostics_After_Publication_Observed : BOOL;
  Output_Projection_Last_Observed : BOOL;
  Runtime_Ownership_Valid : BOOL;
  Diagnostics_Ownership_Valid : BOOL;
  OpenTherm_Ownership_Valid : BOOL;
  Cascade_Ownership_Valid : BOOL;
  Safety_Ownership_Valid : BOOL;
  Observation_Status_Code : UINT;
  Observation_Status_Text : STRING(128);
END_STRUCT;
END_TYPE

TYPE ST_Heating_Runtime_Phase_Event : STRUCT
  Phase : E_Heating_Runtime_Phase;
  Event_Active : BOOL;
  Event_Completed : BOOL;
  Event_Failed : BOOL;
  Start_Time_MS : UDINT;
  End_Time_MS : UDINT;
  Duration_MS : UDINT;
  Ordering_Valid : BOOL;
  Isolation_Valid : BOOL;
  Status_Code : UINT;
  Status_Text : STRING(128);
  Diagnostics_Visible : BOOL;
  Explainability_Visible : BOOL;
  Safety_Integrity_Valid : BOOL;
  OpenTherm_Ownership_Valid : BOOL;
  Cascade_Ownership_Valid : BOOL;
END_STRUCT;
END_TYPE

TYPE ST_Heating_Runtime_Phase_Transition : STRUCT
  Previous_Phase : E_Heating_Runtime_Phase;
  Current_Phase : E_Heating_Runtime_Phase;
  Next_Phase : E_Heating_Runtime_Phase;
  Transition_Active : BOOL;
  Transition_Completed : BOOL;
  Transition_Failed : BOOL;
  Transition_Start_MS : UDINT;
  Transition_End_MS : UDINT;
  Transition_Duration_MS : UDINT;
  Sequencing_Valid : BOOL;
  Ownership_Valid : BOOL;
  Synchronization_Valid : BOOL;
  Status_Code : UINT;
  Status_Text : STRING(128);
END_STRUCT;
END_TYPE

TYPE ST_Heating_Runtime_Predictive_State : STRUCT
  Predictive_Analytics_Visible : BOOL;
  Predictive_Analytics_Degraded : BOOL;
  Predictive_Analytics_Attention : BOOL;
  Runtime_Stable : BOOL;
  Runtime_Stability_Score : UINT;
  Runtime_Degradation_Observation : UINT;
  Runtime_Failure_Observation : UINT;
  Source_Instability_Observation : UINT;
  Source_Instability_Attention : BOOL;
  Source_Oscillation_Trend_Visible : BOOL;
  Source_Degraded_Trend_Visible : BOOL;
  Source_Loss_Trend_Visible : BOOL;
  Cascade_Degradation_Observation : UINT;
  Cascade_Degraded_Trend_Visible : BOOL;
  OpenTherm_Instability_Observation : UINT;
  OpenTherm_Degraded_Trend_Visible : BOOL;
  Sequencing_Observation : UINT;
  Ownership_Observation : UINT;
  Synchronization_Observation : UINT;
  Status_Code : UINT;
  Status_Text : STRING(128);
END_STRUCT;
END_TYPE

TYPE ST_Heating_Runtime_Source_Instability_State : STRUCT
  Visible : BOOL;
  Source_Switch_Count : UINT;
  Fallback_Activation_Count : UINT;
  Fallback_Recovery_Count : UINT;
  Source_Loss_Count : UINT;
  Degraded_Trend_Visible : BOOL;
  Recovery_Trend_Visible : BOOL;
  Oscillation_Detected : BOOL;
  Instability_Attention : BOOL;
  Instability_Score : REAL;
  Confidence_Volatility : REAL;
  Source_Trust_Trend : REAL;
  Status_Code : UINT;
  Status_Text : STRING(128);
  Last_Observation_MS : UDINT;
END_STRUCT;
END_TYPE

TYPE ST_Heating_Runtime_Supervisory_Publication : STRUCT
  Supervisory_Visible : BOOL;
  Predictive_State : ST_Heating_Runtime_Predictive_State;
  Runtime_Degraded : BOOL;
  Runtime_Fault : BOOL;
  Source_Instability_Attention : BOOL;
  Source_Oscillation_Trend_Visible : BOOL;
  Explainability_Degraded : BOOL;
  Diagnostics_Degraded : BOOL;
  Causality_Active : BOOL;
  Propagation_Detected : BOOL;
  Reconstruction_Visible : BOOL;
  Status_Code : UINT;
  Status_Text : STRING(128);
END_STRUCT;
END_TYPE

TYPE ST_Heating_Schedule_Event : STRUCT
  Enabled : BOOL := FALSE;
  Comfort_Time_MS : UDINT := 28800000;
  Weekday_Mask : BYTE := 127;
  Preheat_Boost : REAL := 0.5;
  Adaptive_Enabled : BOOL := TRUE;
  Adaptive_Step_MS : UDINT := 300000;
  Adaptive_Max_Offset_MS : UDINT := 3600000;
END_STRUCT;
END_TYPE

TYPE ST_History_Record : STRUCT
  timestamp_ms : UDINT := 0;
  event_code : WORD := 0;
  event_value : REAL := 0.0;
  unit : BYTE := 0;
  zone_id : BYTE := 0;
  operator_id : STRING(10) := '';
  priority : E_ALERT_PRIORITY := E_ALERT_PRIORITY.ALERT_PRIORITY_NONE;
END_STRUCT;
END_TYPE

TYPE ST_IO_Binding_Record : STRUCT
  Binding_Valid : BOOL;
  Binding_Version : UDINT;
  Physical_Channel_Id : UINT;
  Logical_Device_Id : UINT;
  Domain_Id : UINT;
  Role_Id : UINT;
  Controller_Id : UINT;
  Module_Id : UINT;
  Terminal_Id : UINT;
  Inverted : BOOL;
  Required : BOOL;
  Quality_Required : BOOL;
  Status_Code : UINT;
  Status_Text : STRING(128);
END_STRUCT;
END_TYPE

TYPE ST_Input_Quality_Record : STRUCT
  Quality_Visible : BOOL;
  Value_Valid : BOOL;
  Value_Degraded : BOOL;
  Spike_Detected : BOOL;
  Stuck_Detected : BOOL;
  Confidence : REAL;
  Last_Value : REAL;
  Last_Change_MS : UDINT;
  Reason_Code : UINT;
  Reason_Text : STRING(128);
END_STRUCT;
END_TYPE

TYPE ST_Maintenance_Access_Config : STRUCT
  maintenance_enabled : BOOL := FALSE;
  max_duration_minutes : UDINT := 60;
  requires_two_person : BOOL := TRUE;
  access_level_required : BYTE := 2;
END_STRUCT;
END_TYPE

TYPE ST_Manifold_Status : STRUCT
  Pump_On : BOOL;
  Pump_Current : REAL;
  Pressure : REAL;
  Temp_Supply : REAL;
  Temp_Return : REAL;
  Valve_Pos : REAL;
  Error : BOOL;
  Error_ID : WORD;
  Health : ST_Device_Health;
END_STRUCT;
END_TYPE

TYPE ST_Modbus_RTU_Config : STRUCT
  Port_Name : STRING(32);
  Baudrate : UDINT;
  Parity : BYTE;
  Stop_Bits : BYTE;
  Data_Bits : BYTE;
  Slave_ID : BYTE;
  Poll_Interval_MS : UDINT;
  Request_Timeout_MS : UDINT;
  Retry_Count : INT;
END_STRUCT;
END_TYPE

TYPE ST_Modbus_RTU_Frame : STRUCT
  Valid : BOOL;
  Length : UINT;
  Data : ARRAY[0..255] OF BYTE;
  CRC : WORD;
END_STRUCT;
END_TYPE

TYPE ST_Modbus_Request : STRUCT
  Enable : BOOL;
  Slave_ID : BYTE;
  Function_Code : E_Modbus_Function;
  Start_Register : UINT;
  Register_Count : UINT;
  Write_Value : ARRAY[1..32] OF WORD;
  Sequence : UDINT;
  Timeout_MS : UDINT;
END_STRUCT;
END_TYPE

TYPE ST_Modbus_Response : STRUCT
  Busy : BOOL;
  Done : BOOL;
  Error : BOOL;
  Error_Code : WORD;
  Read_Value : ARRAY[1..32] OF WORD;
  Last_Sequence : UDINT;
  Last_Update_MS : UDINT;
END_STRUCT;
END_TYPE

TYPE ST_OpenTherm_Command : STRUCT
  Enable : BOOL;
  Setpoint_x10 : UINT;
  Sequence : UDINT;
  Last_Write_MS : UDINT;
END_STRUCT;
END_TYPE

TYPE ST_OpenTherm_Register_Map : STRUCT
  Base_Register : UINT;
  Cmd_Enable_Offset : UINT;
  Cmd_Setpoint_x10_Offset : UINT;
  Cmd_Seq_Lo_Offset : UINT;
  Cmd_Seq_Hi_Offset : UINT;
  Status_Heartbeat_Lo_Offset : UINT;
  Status_Heartbeat_Hi_Offset : UINT;
  Status_Ack_Seq_Lo_Offset : UINT;
  Status_Ack_Seq_Hi_Offset : UINT;
  Status_Word_Offset : UINT;
  Error_Code_Offset : UINT;
  Modulation_x10_Offset : UINT;
  Boiler_Temp_x10_Offset : UINT;
END_STRUCT;
END_TYPE

TYPE ST_OpenTherm_Status : STRUCT
  Raw_Heartbeat : UDINT;
  Raw_Ack_Seq : UDINT;
  Raw_Online : BOOL;
  Raw_Error : BOOL;
  Raw_Flame : BOOL;
  Raw_Modulation_x10 : UINT;
  Raw_Boiler_Temp_x10 : INT;
  Raw_Status_Word : WORD;
  Raw_Error_Code : WORD;
  Adapter_Online : BOOL;
  Adapter_Error : BOOL;
  Command_Ack : BOOL;
  Command_Timeout : BOOL;
  Heartbeat_Timeout : BOOL;
  Last_Heartbeat : UDINT;
  Last_Heartbeat_MS : UDINT;
  Heartbeat_Age_MS : UDINT;
  Command_Age_MS : UDINT;
  Last_Command_Ack_Seq : UDINT;
  Adapter_State : E_OpenTherm_Adapter_State;
  Error_State : E_OpenTherm_Error;
END_STRUCT;
END_TYPE

TYPE ST_OpenTherm_Wire_Image : STRUCT
  Cmd_Enable : WORD;
  Cmd_Setpoint_x10 : WORD;
  Cmd_Seq_Lo : WORD;
  Cmd_Seq_Hi : WORD;
  Status_Heartbeat_Lo : WORD;
  Status_Heartbeat_Hi : WORD;
  Status_Ack_Seq_Lo : WORD;
  Status_Ack_Seq_Hi : WORD;
  Status_Word : WORD;
  Error_Code : WORD;
  Modulation_x10 : WORD;
  Boiler_Temp_x10 : WORD;
END_STRUCT;
END_TYPE

TYPE ST_Operator_Zone_Rights : STRUCT
  operator_id : STRING(10);
  global_access_level : BYTE := 0;
  zone_masks : DWORD;
  last_modified : UDINT;
END_STRUCT;
END_TYPE

TYPE ST_Outdoor_Zone_Config : STRUCT
  zone_id : BYTE := 0;
  lighting_circuit_id : BYTE := 0;
  auto_enabled : BOOL := TRUE;
  party_mode_enabled : BOOL := FALSE;
END_STRUCT;
END_TYPE

TYPE ST_Owen_Analog_Value : STRUCT
  rValue : REAL;
  uiCycleTime : UINT;
  wStatus : WORD;
END_STRUCT;
END_TYPE

TYPE ST_Predictive_Diagnostics_State : STRUCT
  Runtime_Valid : BOOL;
  Runtime_System_Time_MS : UDINT;
  Device_Id : UINT;
  Device_Class : UINT;
  Valve_Group_Id : UINT;
  Failure_Count : UINT;
  Timeout_Count : UINT;
  Conflict_Count : UINT;
  Recovery_Denied_Count : UINT;
  Wear_Score : REAL;
  Reliability_Score : REAL;
  Intermittent_Fault_Suspected : BOOL;
  Degradation_Accumulating : BOOL;
  Service_Recommended : BOOL;
  Service_Urgent : BOOL;
  Predictive_Quarantine_Recommended : BOOL;
  Status_Code : UINT;
  Status_Text : STRING(160);
END_STRUCT;
END_TYPE

TYPE ST_Rule : STRUCT
  Action_Type : INT;
  Action_Target_ID : INT;
  Action_Value : REAL;
  Condition_Type : INT;
  Condition_Target_ID : INT;
  Condition_Op : INT;
  Condition_Value : REAL;
  Condition_Value_Max : REAL;
END_STRUCT;
END_TYPE

TYPE ST_Rule_Action : STRUCT
  Active : BOOL;
  Triggered : BOOL;
  Action_Type : E_Rule_Action_Type;
  Target_ID : BYTE;
  Value : REAL;
END_STRUCT;
END_TYPE

TYPE ST_Runtime_Bus_Frame : STRUCT
  Frame_Valid : BOOL;
  Frame_Time_MS : UDINT;
  Frame_Id : UDINT;
  Source_Controller_Id : UINT;
  Source_Runtime_Node_Id : UINT;
  Target_Runtime_Node_Id : UINT;
  Frame_Class : UINT;
  Frame_Sequence_Id : UDINT;
  Frame_Ack_Required : BOOL;
  Frame_Ack_Received : BOOL;
  Authority_State_Frame : BOOL;
  Recovery_State_Frame : BOOL;
  Quarantine_State_Frame : BOOL;
  Topology_State_Frame : BOOL;
  Binding_State_Frame : BOOL;
  Predictive_State_Frame : BOOL;
  Replication_Consistent : BOOL;
  Replication_Stale : BOOL;
  Replication_Rejected : BOOL;
  Status_Code : UINT;
  Status_Text : STRING(160);
END_STRUCT;
END_TYPE

TYPE ST_Runtime_Node_Discovery_State : STRUCT
  Runtime_Valid : BOOL;
  Runtime_System_Time_MS : UDINT;
  Discovery_Active : BOOL;
  Node_Discovered : BOOL;
  Node_Validated : BOOL;
  Node_Authorized : BOOL;
  Node_Quarantined : BOOL;
  Controller_Id : UINT;
  Runtime_Node_Id : UINT;
  Authority_Class : UINT;
  Deployment_Assigned : BOOL;
  Execution_Domain_Assigned : BOOL;
  Capability_Validated : BOOL;
  Discovery_Timeout : BOOL;
  Discovery_Rejected : BOOL;
  Status_Code : UINT;
  Status_Text : STRING(160);
END_STRUCT;
END_TYPE

TYPE ST_Runtime_Node_Session : STRUCT
  Session_Valid : BOOL;
  Session_Id : UDINT;
  Session_Start_MS : UDINT;
  Last_Heartbeat_MS : UDINT;
  Controller_Id : UINT;
  Runtime_Node_Id : UINT;
  Session_Connected : BOOL;
  Session_Stale : BOOL;
  Session_Reconnect_Required : BOOL;
  Session_Quarantined : BOOL;
  Transport_Healthy : BOOL;
  Runtime_Replication_Healthy : BOOL;
  Authority_Granted : BOOL;
  Authority_Revoked : BOOL;
  Status_Code : UINT;
  Status_Text : STRING(160);
END_STRUCT;
END_TYPE

TYPE ST_Runtime_Restart_Continuity_State : STRUCT
  Runtime_Valid : BOOL;
  Runtime_System_Time_MS : UDINT;
  Cold_Start_Detected : BOOL;
  Warm_Restart_Detected : BOOL;
  Restore_Requested : BOOL;
  Restore_Allowed : BOOL;
  Restore_Blocked : BOOL;
  Restore_Completed : BOOL;
  Retained_State_Valid : BOOL;
  Topology_Restore_Valid : BOOL;
  Config_Restore_Valid : BOOL;
  Recovery_Restore_Valid : BOOL;
  Quarantine_Restore_Valid : BOOL;
  Active_Config_Version : UDINT;
  Restored_Config_Version : UDINT;
  Last_Stable_Config_Version : UDINT;
  Post_Restart_Validation_Required : BOOL;
  Post_Restart_Validation_OK : BOOL;
  Post_Restart_Validation_Failed : BOOL;
  Safe_Mode_Required : BOOL;
  Operator_Ack_Required : BOOL;
  Status_Code : UINT;
  Status_Text : STRING(160);
END_STRUCT;
END_TYPE

TYPE ST_Scenario_Config : STRUCT
  scenario_id : E_SCENARIO_TYPE;
  lighting_level_base : BYTE := 100;
  lighting_level_accent : BYTE := 100;
  floor_heating_adjust_celsius : REAL := 0.0;
  ventilation_speed_percent : BYTE := 50;
  sockets_enabled : BOOL := TRUE;
  blinds_position_percent : BYTE := 0;
  Presence_Simulation_Enabled : BOOL := FALSE;
END_STRUCT;
END_TYPE

TYPE ST_Scenario_Stats : STRUCT
  Activations : UDINT;
  Success_Count : UDINT;
  Failure_Count : UDINT;
  Success_Rate : REAL;
  Avg_Result_Value : REAL;
  Stability_Counter : INT;
  Last_Activation : UDINT;
END_STRUCT;
END_TYPE

TYPE ST_Scenario_Transition_Config : STRUCT
  current_scenario : E_SCENARIO_TYPE;
  target_scenario : E_SCENARIO_TYPE;
  min_duration_minutes : UDINT := 5;
  transition_allowed : BOOL := FALSE;
END_STRUCT;
END_TYPE

TYPE ST_Security_Global_Config : STRUCT
  PIN_Code : STRING(4) := '1234';
  Phones : ARRAY[1..GVL_CONSTANTS.C_MAX_SECURITY_PHONES] OF STRING(15);
  entry_delay_seconds : UDINT := 30;
  exit_delay_seconds : UDINT := 60;
  alarm_duration_seconds : UDINT := 180;
  two_person_timeout_seconds : UDINT := 120;
  max_access_attempts : BYTE := 3;
  auto_arm_enabled : BOOL := FALSE;
  auto_arm_time_ms : UDINT := 0;
  enable_2fa : BOOL := TRUE;
  gate_open_pulse_ms : UDINT := GVL_CONSTANTS.C_MS_IN_SECOND;
  wicket_open_pulse_ms : UDINT := GVL_CONSTANTS.C_MS_IN_SECOND;
  lock_open_pulse_ms : UDINT := GVL_CONSTANTS.C_MS_IN_SECOND;
  lock_close_pulse_ms : UDINT := GVL_CONSTANTS.C_MS_IN_SECOND;
  bypass_motion : ARRAY[1..16] OF BOOL;
  bypass_doors : ARRAY[1..GVL_CONSTANTS.C_MAX_DOOR_SENSORS] OF BOOL;
  bypass_windows : ARRAY[1..16] OF BOOL;
END_STRUCT;
END_TYPE

TYPE ST_Security_Zone_State : STRUCT
  Armed : BOOL;
  Alarm : BOOL;
  Bypassed : BOOL;
  Last_Trigger_Time : DT;
  Trigger_Count : UINT;
END_STRUCT;
END_TYPE

TYPE ST_Sensor_Calibration_Record : STRUCT
  sensor_id : UDINT := 0;
  sensor_type : E_SENSOR_TYPE;
  zone_id : BYTE := 0;
  offset : REAL := 0.0;
  multiplier : REAL := 1.0;
  last_calibration_timestamp : UDINT := 0;
  verification_passed : BOOL := FALSE;
END_STRUCT;
END_TYPE

TYPE ST_State_Snapshot : STRUCT
  timestamp_ms : UDINT := 0;
  operator_id : STRING(10) := '';
  scenario_id : E_SCENARIO_TYPE := E_SCENARIO_TYPE.SCENARIO_NONE;
  lighting_levels : ARRAY[1..GVL_CONSTANTS.C_MAX_LIGHTING_ZONES] OF BYTE;
  floor_heating_setpoints : ARRAY[1..GVL_CONSTANTS.C_MAX_HEATING_CIRCUITS] OF REAL;
  alarm_active : BOOL := FALSE;
  crc32 : DWORD := 0;
END_STRUCT;
END_TYPE

TYPE ST_System_Diagnostics : STRUCT
  Freeze_Hardware_Event_Pending : BOOL;
  Freeze_Hardware_Event_Text : STRING(200);
  Backup_Pump_Fault : BOOL;
  Electric_Heater_Fault : BOOL;
  Backup_Pump_Recovered_After_Retry : BOOL;
  Electric_Heater_Recovered_After_Retry : BOOL;
  Backup_Pump_Out_Of_Service : BOOL;
  Electric_Heater_Out_Of_Service : BOOL;
  Pump_Exercise_Active : BOOL;
  Pump_Exercise_Failed : BOOL;
  Pump_Exercise_Last_Equipment : STRING(80);
  Pump_Exercise_Last_Result : STRING(120);
  Pump_Exercise_No_Feedback_Count : INT;
  Manifold_Pump_Exercise_Count : ARRAY[1..GVL_CONSTANTS.C_MAX_MANIFOLDS] OF UDINT;
  DHW_Heating_Pump_Exercise_Count : UDINT;
  DHW_Circ_Pump_Exercise_Count : UDINT;
  Backup_Pump_Exercise_Count : UDINT;
  Pump_Exercise_Event_Seq : UDINT;
  Pump_Exercise_Journal_1 : STRING(200);
  Pump_Exercise_Journal_2 : STRING(200);
  Pump_Exercise_Journal_3 : STRING(200);
  Pump_Exercise_Journal_Last_Seq : UDINT;
  Pump_Maintenance_Required : BOOL;
  Pump_Maintenance_Warning : BOOL;
  Manifold_Pump_Out_Of_Service : ARRAY[1..GVL_CONSTANTS.C_MAX_MANIFOLDS] OF BOOL;
  DHW_Heating_Pump_Out_Of_Service : BOOL;
  DHW_Circ_Pump_Out_Of_Service : BOOL;
  Maintenance_Last_Action : STRING(120);
  Operator_Action_Blocked : BOOL;
  Operator_Block_Reason : STRING(160);
  Operator_Last_Forbidden_Action : STRING(160);
  Operator_Journal_1 : STRING(200);
  Operator_Journal_2 : STRING(200);
  Operator_Journal_3 : STRING(200);
  Operator_Journal_Event_Seq : UDINT;
  Operator_Journal_Last_Seq : UDINT;
  Dangerous_Action_Pending_Confirm : BOOL;
  Dangerous_Action_Confirm_Text : STRING(160);
  Dangerous_Action_Confirm_Deadline_MS : UDINT;
  User_Access_Level_Active : INT;
  User_Access_Denied : BOOL;
  User_Access_Deny_Reason : STRING(160);
  Valve_Test_Mode_Active : BOOL;
  Valve_Test_Deadline_MS : UDINT;
  Valve_Test_Remaining_MS : UDINT;
  Valve_Test_Validation_OK : BOOL;
  Valve_Test_Validation_Text : STRING(160);
  Valve_Test_Forced_Close : BOOL;
  Water_Valve_Test_Mode_Active : BOOL;
  Water_Valve_Test_Deadline_MS : UDINT;
  Water_Valve_Test_Remaining_MS : UDINT;
  Water_Valve_Test_Validation_OK : BOOL;
  Water_Valve_Test_Validation_Text : STRING(160);
  Water_Valve_Test_Forced_Close : BOOL;
  Gas_Valve_Test_Mode_Active : BOOL;
  Gas_Valve_Test_Deadline_MS : UDINT;
  Gas_Valve_Test_Remaining_MS : UDINT;
  Gas_Valve_Test_Validation_OK : BOOL;
  Gas_Valve_Test_Validation_Text : STRING(160);
  Gas_Valve_Test_Forced_Close : BOOL;
  Active_Leak_Sensor_Index : INT;
  Active_Gas_Sensor_Index : INT;
  Active_Leak_Zone_Name : STRING(80);
  Active_Gas_Zone_Name : STRING(80);
  Water_Valve_Test_Context : STRING(160);
  Gas_Valve_Test_Context : STRING(160);
  Water_Recovery_Target_Zone_Index : INT;
  Gas_Recovery_Target_Zone_Index : INT;
  Water_Recovery_Selective_Allowed : BOOL;
  Gas_Recovery_Selective_Allowed : BOOL;
  Water_Recovery_Selective_Text : STRING(160);
  Gas_Recovery_Selective_Text : STRING(160);
  Water_Recovery_Physical_Active : BOOL;
  Water_Recovery_Physical_Zone_Name : STRING(80);
  Water_Zone_Open_Fault : ARRAY[1..32] OF BOOL;
  Water_Zone_Close_Fault : ARRAY[1..32] OF BOOL;
  Water_Valve_Exercise_Last_Zone : INT;
  Water_Valve_Exercise_Last_Result : STRING(160);
  Water_Zone_Critical_Close_Fault : ARRAY[1..32] OF BOOL;
  Water_Close_Fault_Active : BOOL;
  Water_Close_Fault_Zone_Name : STRING(80);
  Water_Close_Fault_Text : STRING(200);
  Water_Zone_Close_Retry_Active : ARRAY[1..32] OF BOOL;
  Water_Zone_Close_Retry_Count : ARRAY[1..32] OF INT;
  Water_Zone_Close_Recovered_After_Retry : ARRAY[1..32] OF BOOL;
  Water_Localization_Failed : BOOL;
  Water_Main_Shutdown_Recommended : BOOL;
  Water_Escalation_Text : STRING(200);
  Alarm_Event_Pulse : BOOL;
  Alarm_Event_Code : UDINT;
  Alarm_Event_Value : REAL;
  Sensor_Fault : BOOL;
  IO_Offline : BOOL;
  Subsystem_Degraded : BOOL;
  Manifold_Pressure_Fault : ARRAY[1..GVL_CONSTANTS.C_MAX_MANIFOLDS] OF BOOL;
  Manifold_Pressure_Diag_Code : ARRAY[1..GVL_CONSTANTS.C_MAX_MANIFOLDS] OF WORD;
  Manifold_Pressure_Fault_Active : BOOL;
  Manifold_Pressure_First_Fault_Index : INT;
  Manifold_Pressure_Fault_Text : STRING(160);
  Manifold_Current_Fault : ARRAY[1..GVL_CONSTANTS.C_MAX_MANIFOLDS] OF BOOL;
  Manifold_Current_Diag_Code : ARRAY[1..GVL_CONSTANTS.C_MAX_MANIFOLDS] OF WORD;
  Manifold_Current_Fault_Active : BOOL;
  Manifold_Current_First_Fault_Index : INT;
  Manifold_Current_Fault_Text : STRING(160);
  Manifold_Return_Temp_Fault : ARRAY[1..GVL_CONSTANTS.C_MAX_MANIFOLDS] OF BOOL;
  Manifold_Return_Temp_Diag_Code : ARRAY[1..GVL_CONSTANTS.C_MAX_MANIFOLDS] OF WORD;
  Manifold_Return_Temp_Fault_Active : BOOL;
  Manifold_Return_Temp_First_Fault_Index : INT;
  Manifold_Return_Temp_Fault_Text : STRING(160);
  Manifold_Sensor_Fault_Count : ARRAY[1..GVL_CONSTANTS.C_MAX_MANIFOLDS] OF INT;
  Manifold_Sensor_Out_Of_Service : ARRAY[1..GVL_CONSTANTS.C_MAX_MANIFOLDS] OF BOOL;
  Manifold_Sensor_Out_Of_Service_Active : BOOL;
  Manifold_Sensor_First_OOS_Index : INT;
  Manifold_Sensor_OOS_Text : STRING(160);
END_STRUCT;
END_TYPE

TYPE ST_System_State_Snapshot : STRUCT
  System_Time_MS : UDINT;
  Current_Scenario : E_SCENARIO_TYPE;
  Security_Armed : BOOL;
  Active_Alarms : INT;
  Zone_Valves : ARRAY[1..GVL_CONSTANTS.C_MAX_HEATING_CIRCUITS] OF BOOL;
  Manifold_Pumps : ARRAY[1..GVL_CONSTANTS.C_MAX_MANIFOLDS] OF BOOL;
  Lighting_States : ARRAY[1..32] OF BYTE;
  Blinds_Positions : ARRAY[1..GVL_CONSTANTS.C_MAX_BLINDS] OF BYTE;
  Socket_States : ARRAY[1..GVL_CONSTANTS.C_MAX_SOCKETS] OF BOOL;
  Gas_Valve_Closed : BOOL;
  Water_Valves_Closed : BOOL;
  Version : UDINT;
END_STRUCT;
END_TYPE

TYPE ST_System_State_Summary : STRUCT
  Outdoor_Temp : REAL;
  Indoor_Temp : ARRAY[1..GVL_CONSTANTS.C_MAX_CLIMATE_ZONES] OF REAL;
  Floor_Temps : ARRAY[1..GVL_CONSTANTS.C_MAX_HEATING_CIRCUITS] OF REAL;
  Humidity : ARRAY[1..GVL_CONSTANTS.C_MAX_HUMIDITY_SENSORS] OF REAL;
  CO2 : ARRAY[1..GVL_CONSTANTS.C_MAX_CO2_SENSORS] OF REAL;
  Gas_Alarm : BOOL;
  Flood_Alarm : BOOL;
  Fire_Alarm : BOOL;
  Security_Alarm : BOOL;
  Security_Armed : BOOL;
END_STRUCT;
END_TYPE

TYPE ST_Tariff_Config : STRUCT
  Enabled : BOOL := FALSE;
  Night_Start_Hour : UINT := 23;
  Night_End_Hour : UINT := 7;
  Boost_Delta : REAL := 2.0;
END_STRUCT;
END_TYPE

TYPE ST_Trace_Entry : STRUCT
  Timestamp_MS : UDINT;
  Layer : E_Trace_Layer;
  Source : E_Trace_Source;
  Reason_Code : E_System_Reason_Code;
  Value_Bool : BOOL;
  Value_Real : REAL;
  Text : STRING(120);
END_STRUCT;
END_TYPE

TYPE ST_Trend_Config : STRUCT
  param_type : BYTE;
  zone_id : BYTE;
  enabled : BOOL;
  deviation_threshold_percent : REAL := 10.0;
  history_days : UDINT := 7;
END_STRUCT;
END_TYPE

TYPE ST_Trend_Data : STRUCT
  config : ST_Trend_Config;
  record_count : UDINT;
  write_index : UDINT;
  sum_values : REAL;
  values : ARRAY[1..100] OF REAL;
  timestamps : ARRAY[1..100] OF UDINT;
  crc32 : DWORD;
END_STRUCT;
END_TYPE

TYPE ST_Trend_Header : STRUCT
  parameter_type : BYTE;
  zone_id : BYTE := 0;
  records_count : UDINT := 0;
  average_value : REAL := 0.0;
  min_value : REAL := 0.0;
  max_value : REAL := 0.0;
END_STRUCT;
END_TYPE

TYPE ST_Trend_History_Record : STRUCT
  timestamp_ms : UDINT := 0;
  value : REAL := 0.0;
END_STRUCT;
END_TYPE

TYPE ST_TwoFactor_Auth_State : STRUCT
  Auth_Method : E_TwoFactor_Method;
  is_pending : BOOL;
  Attempts_Left : UINT;
  Time_Left_S : UINT;
  Is_Success : BOOL;
  Is_Locked : BOOL;
END_STRUCT;
END_TYPE

TYPE ST_TwoFactor_Data : STRUCT
  operator_id : STRING(10);
  AuthMethod : BYTE;
  rfid_tag : STRING(20);
  totp_secret : STRING(32);
  last_modified : UDINT;
END_STRUCT;
END_TYPE

TYPE ST_User_Rule : STRUCT
  Enabled : BOOL;
  Condition_Type : E_Rule_Condition_Type;
  Condition_Target_ID : BYTE;
  Condition_Op : E_Rule_Comparison;
  Condition_Value : REAL;
  Condition_Value_Max : REAL;
  Action_Target_ID : BYTE;
  Action_Value : REAL;
  Action_Type : E_Rule_Action_Type;
  Priority : BYTE;
END_STRUCT;
END_TYPE

TYPE ST_Valve_Test_Config : STRUCT
  valve_id : BYTE := 0;
  test_interval_days : UDINT := 7;
  Nominal_Current : REAL := 0.5;
  nominal_close_time_sec : REAL := 10.0;
  enabled : BOOL := TRUE;
END_STRUCT;
END_TYPE

TYPE ST_Ventilation_Config : STRUCT
  CO2_Threshold : REAL := 800.0;
  Humidity_Threshold : REAL := 65.0;
  Night_Mode_Start : TOD := TOD#23:00;
  Night_Mode_End : TOD := TOD#07:00;
END_STRUCT;
END_TYPE

TYPE ST_Ventilation_Global_Config : STRUCT
  enable_ventilation : BOOL := TRUE;
  total_units : BYTE := 8;
  default_supply_speed : BYTE := 40;
  default_exhaust_speed : BYTE := 40;
  Degraded_Exhaust_Limit : BYTE := 30;
  Scenario_Modes : ARRAY[1..GVL_CONSTANTS.C_MAX_SCENARIOS] OF ST_Ventilation_Scenario_Mode;
  wet_zone_to_exhaust_map : ARRAY[1..GVL_CONSTANTS.C_MAX_WET_ZONES] OF INT := [2, 3, 4, 5];
  pv3_exhaust_index : INT := 3;
END_STRUCT;
END_TYPE

TYPE ST_Ventilation_Scenario_Mode : STRUCT
  Scenario_ID : BYTE;
  Scenario_Priority : BYTE;
  Fire_Alarm : BOOL;
  Methane_Alarm : BOOL;
  Smoke_Detected : BOOL;
  Exhaust_Modes : ARRAY[1..GVL_CONSTANTS.C_MAX_EXHAUST_FANS] OF BYTE;
  Supply_Modes : ARRAY[1..GVL_CONSTANTS.C_MAX_SUPPLY_FANS] OF BYTE;
  Base_Fan_Speed : BYTE := 50;
  Target_Temp : REAL := 22.0;
END_STRUCT;
END_TYPE

TYPE ST_Ventilation_Unit : STRUCT
  Enabled : BOOL;
  Speed_Percent : REAL;
  Filter_Dirty : BOOL;
  Error : BOOL;
  Mode : BYTE;
END_STRUCT;
END_TYPE

TYPE ST_Ventilation_Unit_Config : STRUCT
  unit_id : BYTE := 0;
  unit_type : E_VENTILATION_UNIT_TYPE;
  location : E_VENTILATION_LOCATION;
  min_speed : BYTE := 20;
  max_speed : BYTE := 100;
  Threshold_Hum : REAL := 65.0;
  has_smoke_detector : BOOL := FALSE;
END_STRUCT;
END_TYPE

TYPE ST_Water_Actuator_Diagnostics_State : STRUCT
  Runtime_Valid : BOOL;
  Runtime_System_Time_MS : UDINT;
  Valve_Group_Id : UINT;
  Travel_Active : BOOL;
  Travel_Timeout : BOOL;
  Stuck_Suspected : BOOL;
  Intermittent_Failure_Suspected : BOOL;
  Travel_Time_MS : UDINT;
  Failure_Count : UINT;
  Diagnostics_Degraded : BOOL;
  Escalation_Required : BOOL;
  Status_Code : UINT;
  Status_Text : STRING(128);
END_STRUCT;
END_TYPE

TYPE ST_Water_Event_Log_Record : STRUCT
  Runtime_Valid : BOOL; Event_Time_MS : UDINT; Event_Id : UINT; Event_Text : STRING(80);
END_STRUCT;
END_TYPE

TYPE ST_Water_Graph_Traversal_State : STRUCT
  Runtime_Valid : BOOL;
  Runtime_System_Time_MS : UDINT;
  Sensor_Id : UINT;
  Start_Segment_Id : UINT;
  Target_Valve_Group_Id : UINT;
  Upstream_Dependency_Detected : BOOL;
  Downstream_Impact_Detected : BOOL;
  Shared_Trunk_Traversal : BOOL;
  Traversal_Valid : BOOL;
  Traversal_Conflict : BOOL;
  Traversal_Ambiguous : BOOL;
  Dependency_Depth : UINT;
  Selective_Path_Allowed : BOOL;
  Global_Fallback_Required : BOOL;
  Status_Code : UINT;
  Status_Text : STRING(128);
END_STRUCT;
END_TYPE

TYPE ST_Water_Hydraulic_Isolation_Group : STRUCT
  Runtime_Valid : BOOL;
  Isolation_Group_Id : UINT;
  Valve_Group_Id : UINT;
  Fallback_Domain_Id : UINT;
  Shared_Segment_Count : UINT;
  Shared_Sensor_Count : UINT;
  Isolation_Valid : BOOL;
  Isolation_Ambiguous : BOOL;
  Selective_Isolation_Allowed : BOOL;
  Global_Fallback_Required : BOOL;
  Status_Code : UINT;
  Status_Text : STRING(128);
END_STRUCT;
END_TYPE

TYPE ST_Water_Hydraulic_Topology_Edge : STRUCT
  Runtime_Valid : BOOL;
  Edge_Id : UINT;
  Upstream_Segment_Id : UINT;
  Downstream_Segment_Id : UINT;
  Isolation_Group_Id : UINT;
  Valve_Group_Id : UINT;
  Shared_Trunk : BOOL;
  Cross_Zone_Dependency : BOOL;
  Dependency_Valid : BOOL;
  Dependency_Ambiguous : BOOL;
  Selective_Isolation_Allowed : BOOL;
  Global_Fallback_Required : BOOL;
  Status_Code : UINT;
  Status_Text : STRING(128);
END_STRUCT;
END_TYPE

TYPE ST_Water_Hydraulic_Topology_Node : STRUCT
  Runtime_Valid : BOOL;
  Sensor_Id : UINT;
  Hydraulic_Zone_Id : UINT;
  Hydraulic_Segment_Id : UINT;
  Isolation_Group_Id : UINT;
  Valve_Group_Id : UINT;
  Fallback_Domain_Id : UINT;
  Mapping_Valid : BOOL;
  Mapping_Ambiguous : BOOL;
  Shared_Valve_Group : BOOL;
  Selective_Isolation_Allowed : BOOL;
  Global_Fallback_Required : BOOL;
  Status_Code : UINT;
  Status_Text : STRING(128);
END_STRUCT;
END_TYPE

TYPE ST_Water_Isolation_Authority_State : STRUCT
  Decision_Valid : BOOL;
  Decision_System_Time_MS : UDINT;
  Isolation_Requested : BOOL;
  Selective_Candidate : BOOL;
  Global_Fallback_Candidate : BOOL;
  Selective_Authority_Allowed : BOOL;
  Global_Fallback_Required : BOOL;
  Authority_Denied : BOOL;
  Hydraulic_Zone_Id : UINT;
  Isolation_Group_Id : UINT;
  Valve_Group_Id : UINT;
  Mapping_Valid : BOOL;
  Deterministic_Target_Valid : BOOL;
  Safety_Context_Allows_Selective : BOOL;
  Valve_Diagnostics_Available : BOOL;
  Valve_Confirmation_Required : BOOL;
  Active_Global_Close_Path : BOOL;
  Active_Safety_Latch : BOOL;
  Decision_Code : UINT;
  Decision_Text : STRING(128);
  Authority_Selected_Event : BOOL;
  Authority_Denied_Event : BOOL;
  Fallback_Selected_Event : BOOL;
END_STRUCT;
END_TYPE

TYPE ST_Water_Isolation_Path_Runtime_State : STRUCT
  Runtime_Valid : BOOL;
  Runtime_System_Time_MS : UDINT;
  Sensor_Id : UINT;
  Isolation_Path_Valid : BOOL;
  Isolation_Path_Ambiguous : BOOL;
  Multi_Valve_Path : BOOL;
  Active_Isolation_Group_Id : UINT;
  Active_Valve_Group_Id : UINT;
  Shared_Trunk_Impact : BOOL;
  Cross_Zone_Impact : BOOL;
  Selective_Isolation_Allowed : BOOL;
  Global_Fallback_Required : BOOL;
  Conflict_Detected : BOOL;
  Status_Code : UINT;
  Status_Text : STRING(128);
END_STRUCT;
END_TYPE

TYPE ST_Water_Isolation_Runtime_State : STRUCT
  Projection_Valid : BOOL;
  Projection_System_Time_MS : UDINT;
  Isolation_Requested : BOOL;
  Selective_Isolation_Requested : BOOL;
  Global_Isolation_Requested : BOOL;
  Hydraulic_Zone_Id : UINT;
  Isolation_Group_Id : UINT;
  Valve_Group_Id : UINT;
  Mapping_Valid : BOOL;
  Fallback_To_Global_Required : BOOL;
  Active_Global_Close_Path : BOOL;
  Active_Safety_Latch : BOOL;
  Reason_Code : UINT;
  Reason_Text : STRING(128);
  Isolation_Requested_Event : BOOL;
  Fallback_To_Global_Event : BOOL;
  Supervisory_Observation_Only : BOOL;
END_STRUCT;
END_TYPE

TYPE ST_Water_Leak_Runtime_State : STRUCT
  Projection_Valid : BOOL;
  Projection_System_Time_MS : UDINT;
  Physical_Sensor_Index : UINT;
  Physical_Input_Valid : BOOL;
  Logical_Sensor_Valid : BOOL;
  Leak_Warning_Active : BOOL;
  Leak_Confirmed : BOOL;
  Leak_Cleared : BOOL;
  Leak_Degraded : BOOL;
  Hydraulic_Zone_Id : UINT;
  Hydraulic_Segment_Id : UINT;
  Isolation_Group_Id : UINT;
  Valve_Group_Id : UINT;
  Mapping_Valid : BOOL;
  Mapping_Missing : BOOL;
  Selective_Isolation_Possible : BOOL;
  Fallback_Global_Isolation_Required : BOOL;
  Leak_Confidence : REAL;
  Sensor_Quality_Valid : BOOL;
  Sensor_Stuck_Suspected : BOOL;
  Sensor_Noise_Suspected : BOOL;
  Reason_Code : UINT;
  Reason_Text : STRING(128);
  Warning_Started_Event : BOOL;
  Leak_Confirmed_Event : BOOL;
  Leak_Cleared_Event : BOOL;
  Isolation_Requested_Event : BOOL;
  Mapping_Invalid_Event : BOOL;
  Active_Safety_Leak_Latched : BOOL;
  Active_Global_Close_Path : BOOL;
  Supervisory_Observation_Only : BOOL;
END_STRUCT;
END_TYPE

TYPE ST_Water_Orchestration_Runtime_State : STRUCT
  Runtime_Valid : BOOL;
  Runtime_System_Time_MS : UDINT;
  Isolation_Sequence_Active : BOOL;
  Recovery_Sequence_Active : BOOL;
  Staged_Close_Required : BOOL;
  Staged_Open_Required : BOOL;
  Shared_Trunk_Sequencing : BOOL;
  Rollback_Required : BOOL;
  Escalation_Required : BOOL;
  Observation_Window_Active : BOOL;
  Sequencing_Valid : BOOL;
  Status_Code : UINT;
  Status_Text : STRING(128);
END_STRUCT;
END_TYPE

TYPE ST_Water_Output_Projection_State : STRUCT
  Projection_Valid : BOOL;
  Projection_System_Time_MS : UDINT;
  Output_Owner_Valid : BOOL;
  Output_Owner_Id : UINT;
  Valve_Id : UINT;
  Valve_Group_Id : UINT;
  Selective_Authority_Allowed : BOOL;
  Global_Fallback_Required : BOOL;
  Authority_Valid : BOOL;
  Physical_Close_Project : BOOL;
  Physical_Open_Project : BOOL;
  Expected_Closed : BOOL;
  Expected_Open : BOOL;
  Confirmed_Closed : BOOL;
  Confirmed_Open : BOOL;
  Confirmation_Unknown : BOOL;
  Projection_Allowed : BOOL;
  Projection_Denied : BOOL;
  Projection_Code : UINT;
  Projection_Text : STRING(128);
  Projection_Activated_Event : BOOL;
  Projection_Denied_Event : BOOL;
END_STRUCT;
END_TYPE

TYPE ST_Water_Output_Reconciliation_State : STRUCT
  Runtime_Valid : BOOL;
  Runtime_System_Time_MS : UDINT;
  Valve_Group_Id : UINT;
  Projection_Active : BOOL;
  Runtime_Output_Active : BOOL;
  Expected_Closed : BOOL;
  Confirmed_Closed : BOOL;
  Confirmation_Unknown : BOOL;
  Reconciliation_Healthy : BOOL;
  Projection_Runtime_Mismatch : BOOL;
  Projection_Confirmation_Mismatch : BOOL;
  Conflict_Detected : BOOL;
  Topology_Invalid : BOOL;
  Status_Code : UINT;
  Status_Text : STRING(128);
END_STRUCT;
END_TYPE

TYPE ST_Water_Physical_Convergence_State : STRUCT
  Runtime_Valid : BOOL;
  Runtime_System_Time_MS : UDINT;
  Sensor_Id : UINT;
  Projection_Active : BOOL;
  Physical_State_Confirmed : BOOL;
  Runtime_Converged : BOOL;
  Physical_Open_Confirmed : BOOL;
  Physical_Closed_Confirmed : BOOL;
  Projection_Mismatch : BOOL;
  Runtime_Mismatch : BOOL;
  Physical_Mismatch : BOOL;
  Convergence_Degraded : BOOL;
  Escalation_Required : BOOL;
  Status_Code : UINT;
  Status_Text : STRING(128);
END_STRUCT;
END_TYPE

TYPE ST_Water_Recovery_FSM_State : STRUCT
  Runtime_Valid : BOOL;
  Runtime_System_Time_MS : UDINT;
  Recovery_Domain_Id : UINT;
  Recovery_Requested : BOOL;
  Recovery_Sequencing_Active : BOOL;
  Recovery_Verification_Window_Active : BOOL;
  Rollback_Required : BOOL;
  Escalation_Required : BOOL;
  Operator_Ack_Required : BOOL;
  Recovery_Completed : BOOL;
  Recovery_Denied : BOOL;
  FSM_State : UINT;
  Status_Code : UINT;
  Status_Text : STRING(128);
END_STRUCT;
END_TYPE

TYPE ST_Water_Recovery_Runtime_State : STRUCT
  Runtime_Valid : BOOL;
  Runtime_System_Time_MS : UDINT;
  Recovery_Requested : BOOL;
  Recovery_Allowed : BOOL;
  Recovery_Denied : BOOL;
  Observation_Window_Active : BOOL;
  Unsafe_Recovery_Detected : BOOL;
  Valve_Degraded : BOOL;
  Confirmation_Healthy : BOOL;
  Recovery_Target_Valid : BOOL;
  Status_Code : UINT;
  Status_Text : STRING(128);
END_STRUCT;
END_TYPE

TYPE ST_Water_Topology_Config_Record : STRUCT
  Config_Valid : BOOL;
  Config_Version : UDINT;
  Sensor_Id : UINT;
  Logical_Zone_Id : UINT;
  Hydraulic_Segment_Id : UINT;
  Isolation_Group_Id : UINT;
  Primary_Valve_Group_Id : UINT;
  Secondary_Valve_Group_Id : UINT;
  Fallback_Domain_Id : UINT;
  Shared_Trunk : BOOL;
  Cross_Zone_Dependency : BOOL;
  Multi_Valve_Required : BOOL;
  Recovery_Domain_Id : UINT;
  Recovery_Requires_Manual_Ack : BOOL;
  Status_Code : UINT;
  Status_Text : STRING(128);
END_STRUCT;
END_TYPE

TYPE ST_Water_Topology_Validation_State : STRUCT
  Runtime_Valid : BOOL;
  Runtime_System_Time_MS : UDINT;
  Sensor_Id : UINT;
  Topology_Valid : BOOL;
  Topology_Ambiguous : BOOL;
  Isolation_Path_Valid : BOOL;
  Shared_Valve_Group : BOOL;
  Missing_Valve_Group : BOOL;
  Invalid_Isolation_Group : BOOL;
  Selective_Isolation_Allowed : BOOL;
  Global_Fallback_Required : BOOL;
  Status_Code : UINT;
  Status_Text : STRING(128);
END_STRUCT;
END_TYPE

TYPE ST_Water_Valve_Feedback_State : STRUCT
  Runtime_Valid : BOOL;
  Runtime_System_Time_MS : UDINT;
  Valve_Group_Id : UINT;
  Feedback_Available : BOOL;
  Physical_Open_Feedback : BOOL;
  Physical_Closed_Feedback : BOOL;
  Confirmed_Open : BOOL;
  Confirmed_Closed : BOOL;
  Feedback_Invalid : BOOL;
  Feedback_Conflict : BOOL;
  Feedback_Timeout : BOOL;
  Travel_Timeout_Active : BOOL;
  Valve_Stuck_Suspected : BOOL;
  Valve_Degraded : BOOL;
  Status_Code : UINT;
  Status_Text : STRING(128);
END_STRUCT;
END_TYPE

TYPE ST_Water_Valve_Runtime_State : STRUCT
  Runtime_Valid : BOOL;
  Runtime_System_Time_MS : UDINT;
  Valve_Id : UINT;
  Valve_Group_Id : UINT;
  Close_Requested : BOOL;
  Open_Requested : BOOL;
  Global_Fallback_Request : BOOL;
  Selective_Authority_Allowed : BOOL;
  Physical_Output_Active : BOOL;
  Output_Command_Projected : BOOL;
  Confirmation_Available : BOOL;
  Confirmed_Open : BOOL;
  Confirmed_Closed : BOOL;
  Confirmation_Timeout : BOOL;
  Confirmation_Unknown : BOOL;
  Diagnostics_Available : BOOL;
  Valve_Healthy : BOOL;
  Valve_Stuck_Suspected : BOOL;
  Travel_Time_Degraded : BOOL;
  Current_Deviation_Detected : BOOL;
  Valve_Degraded : BOOL;
  Unsafe_Reopen_Denied : BOOL;
  Recovery_Allowed : BOOL;
  Status_Code : UINT;
  Status_Text : STRING(128);
  Close_Command_Event : BOOL;
  Open_Command_Event : BOOL;
  Confirmation_Lost_Event : BOOL;
  Valve_Degraded_Event : BOOL;
END_STRUCT;
END_TYPE

TYPE ST_Zone_Adapt_State : STRUCT
  Zone_Weight : REAL;
  Confidence : REAL;
  Activations : UDINT;
  Success_Count : UDINT;
  Failure_Count : UDINT;
  Success_Rate : REAL;
  Avg_Result_Value : REAL;
  Last_Update_MS : UDINT;
END_STRUCT;
END_TYPE

TYPE ST_Zone_Sensors : STRUCT
  Temp_Room : REAL;
  Temp_Floor : REAL;
  Motion_Active : BOOL;
  Switch_Physical : BOOL;
  Light_State : BOOL;
  Maintenance : ST_Component_Maintenance;
END_STRUCT;
END_TYPE

VAR_GLOBAL  (* GVL_AUTHORITY_RESURRECTION_BOUNDARY_FABRIC *)
  Authority_Resurrection_Boundary_Valid : BOOL := FALSE;
  Authority_Resurrection_Bounded : BOOL := FALSE;
  Authority_Recovery_Lineage_Stable : BOOL := FALSE;
  Distributed_Authority_Recovery_Consensus : BOOL := FALSE;
  Authority_Resurrection_Causality_Valid : BOOL := FALSE;
  Resurrection_Timeline_Monotonic : BOOL := FALSE;
  Partial_Recovery_Authority_Leak : BOOL := FALSE;
  Unsafe_Authority_Resurrection_Detected : BOOL := FALSE;
  Resurrection_Authority_Fork_Detected : BOOL := FALSE;
  Authority_Resurrection_Epoch : UDINT := 0;
END_VAR

VAR_GLOBAL  (* GVL_GOVERNANCE_PUBLICATION_BINDING_FABRIC *)
  Governance_Publication_Binding_Valid : BOOL := FALSE;
  Governance_Publication_Binding_Granted : BOOL := FALSE;
  Governance_Publication_Binding_Quarantine_Active : BOOL := TRUE;
  Observability_Publication_Causality_Valid : BOOL := FALSE;
  Upstream_Governance_Lease_Fresh : BOOL := FALSE;
  Governance_Publication_Epoch_Coherent : BOOL := FALSE;
  Publication_Quarantine_Propagation_Valid : BOOL := FALSE;
  Canonical_Observability_Reality_Consistent : BOOL := FALSE;
  Diagnostics_Publication_Consistency_Valid : BOOL := FALSE;
  HMI_Publication_State_Aligned : BOOL := FALSE;
  Blackbox_Invalidation_Lineage_Valid : BOOL := FALSE;
  Distributed_Publication_Consensus_Valid : BOOL := FALSE;
  Stale_Valid_Publication_Detected : BOOL := FALSE;
  LeaseExpired_Governance_Published_As_Healthy : BOOL := FALSE;
  Quarantine_State_Publication_Bypass : BOOL := FALSE;
  Governance_Invalidation_Hidden_From_Observability : BOOL := FALSE;
  Distributed_Publication_State_Fork_Detected : BOOL := FALSE;
  Historical_Invalidation_Causality_Lost : BOOL := FALSE;
  Governance_Publication_Binding_Epoch : UDINT := 0;
  Governance_Publication_Binding_Epoch_Coherent_Runtime : BOOL := FALSE;
  Governance_Publication_Binding_Last_Update_MS : UDINT := 0;
  Governance_Publication_Binding_Lease_Expired : BOOL := TRUE;
  Governance_Publication_Binding_Last_Error_Code : UDINT := 0;
  Governance_Publication_Binding_Last_Error_Text : STRING(160) := '';
  Governance_Publication_Binding_Invalidation_Count : UDINT := 0;
END_VAR

VAR_GLOBAL  (* GVL_OUTPUT_EPOCH *)
  Output_Publication_Epoch : ULINT := 0;
  Output_Publication_Valid : BOOL := FALSE;
  Output_Publication_Allowed : BOOL := TRUE;
  Output_Lease_Active : BOOL := FALSE;
  Output_Lease_Expired : BOOL := FALSE;
  Output_Lease_Timeout_MS : UDINT := 3000;
  Output_Last_Publication_MS : UDINT := 0;
  Output_Last_Refresh_MS : UDINT := 0;
  Output_Last_Invalidation_MS : UDINT := 0;
  Output_Runtime_Epoch : ULINT := 0;
  Output_Runtime_Epoch_Valid : BOOL := FALSE;
  Output_Stale_Detected : BOOL := FALSE;
  Output_Forced_Safe_Decay : BOOL := FALSE;
  Output_Semantic_Continuity_Warning : BOOL := FALSE;
  Output_Last_Error_Code : UDINT := 0;
  Output_Last_Error_Text : STRING(160) := '';
END_VAR

VAR_GLOBAL  (* GVL_OBSERVABILITY_AUTHORITY_FABRIC *)
  Observability_Authority_Valid : BOOL := FALSE;
  Observability_Quarantine_Active : BOOL := TRUE;
  Observability_Publication_Allowed : BOOL := FALSE;
  HMI_Authority_Coherent : BOOL := FALSE;
  Diagnostics_Authority_Coherent : BOOL := FALSE;
  Blackbox_Authority_Coherent : BOOL := FALSE;
  Trend_Authority_Coherent : BOOL := FALSE;
  Alarm_Authority_Coherent : BOOL := FALSE;
  Stale_HMI_State_Detected : BOOL := FALSE;
  Diagnostic_Epoch_Skew_Detected : BOOL := FALSE;
  Post_Revocation_Observability_Lag : BOOL := FALSE;
  Nonauthoritative_Operator_State_Detected : BOOL := FALSE;
  Observability_Epoch : UDINT := 0;
  Observability_Epoch_Coherent : BOOL := FALSE;
  Observability_Last_Update_MS : UDINT := 0;
  Observability_Lease_Expired : BOOL := TRUE;
  Observability_Last_Error_Code : UDINT := 0;
  Observability_Last_Error_Text : STRING(160) := '';
  Observability_Invalidation_Count : UDINT := 0;
END_VAR

{attribute 'qualified_only'}
VAR_GLOBAL  (* GVL_Config_Activation *)
  G_Requested_Config_Version : UDINT;
  G_Staged_Config_Version : UDINT;
  G_Last_Stable_Config_Version : UDINT;
  G_Activation_Request : BOOL;
  G_Rollback_Request : BOOL;
END_VAR

VAR_GLOBAL  (* GVL_PROOF_CONTINUITY_AUDIT_FABRIC *)
  Proof_Continuity_Audit_Active : BOOL := TRUE;
  Proof_Continuity_Observed : BOOL := FALSE;
  Proof_Lineage_Coherent : BOOL := FALSE;
  Proof_Historical_Integrity_Observed : BOOL := FALSE;
  Proof_Audit_ReadOnly_Mode : BOOL := TRUE;
  Proof_Audit_NoTopologyMutation : BOOL := TRUE;
  Proof_Gap_Observed : BOOL := FALSE;
  Proof_Lineage_Drift_Observed : BOOL := FALSE;
  Proof_Consistency_Decay_Observed : BOOL := FALSE;
  Proof_Continuity_Audit_Epoch : UDINT := 0;
END_VAR

VAR_GLOBAL  (* GVL_PHYSICAL_REALITY_VERIFICATION_FABRIC *)
  Physical_Reality_Verification_Active : BOOL := TRUE;
  Physical_Reality_Verification_ReadOnly : BOOL := TRUE;
  Physical_Reality_Verification_NoMutation : BOOL := TRUE;
  Commanded_State_Verified_Physically : BOOL := FALSE;
  Physical_Response_Coherent : BOOL := FALSE;
  Sensor_Physics_Coherent : BOOL := FALSE;
  Physical_Runtime_Reality_Valid : BOOL := FALSE;
  Physical_Reality_Divergence_Detected : BOOL := FALSE;
  Commanded_State_Mismatch_Detected : BOOL := FALSE;
  Impossible_Physical_Response_Detected : BOOL := FALSE;
  Sensor_Physics_Contradiction_Detected : BOOL := FALSE;
  Passive_Physics_Reasoning_Active : BOOL := TRUE;
  Physical_Contradiction_Observed : BOOL := FALSE;
  Physical_Reality_Verification_Epoch : UDINT := 0;
END_VAR

VAR_GLOBAL  (* GVL_PASSIVE_RUNTIME_VERIFICATION_FABRIC *)
  Passive_Runtime_Verification_Active : BOOL := TRUE;
  Runtime_Verification_Consistency_Valid : BOOL := FALSE;
  Runtime_Verification_Lineage_Coherent : BOOL := FALSE;
  Runtime_Verification_Timeline_Monotonic : BOOL := FALSE;
  Passive_Runtime_Verification_ReadOnly : BOOL := TRUE;
  Passive_Runtime_Verification_NoMutation : BOOL := TRUE;
  Passive_Runtime_Verification_NoAuthority : BOOL := TRUE;
  Passive_Runtime_Verification_NoBlocking : BOOL := TRUE;
  Runtime_Semantic_Drift_Observed : BOOL := FALSE;
  Runtime_Consistency_Decay_Observed : BOOL := FALSE;
  Runtime_Verification_Anomaly_Observed : BOOL := FALSE;
  Passive_Runtime_Verification_Epoch : UDINT := 0;
END_VAR

VAR_GLOBAL  (* GVL_HISTORICAL_TRUTH *)
  Historical_Truth_Valid : BOOL := FALSE;
  Historical_Truth_Granted : BOOL := FALSE;
  Historical_Truth_Quarantine_Active : BOOL := TRUE;
  Trend_History_Causally_Immutable : BOOL := FALSE;
  Alarm_Chronology_Immutable : BOOL := FALSE;
  Blackbox_Snapshot_Immutable : BOOL := FALSE;
  Diagnostics_History_Coherent : BOOL := FALSE;
  Failover_Chronology_Coherent : BOOL := FALSE;
  Persisted_Epochs_Coherent : BOOL := FALSE;
  Recovery_Replay_Coherent : BOOL := FALSE;
  Historical_Snapshot_Coherent : BOOL := FALSE;
  Mixed_Authority_Persistence_Absent : BOOL := FALSE;
  History_Epoch_Skew_Detected : BOOL := FALSE;
  Failover_Chronology_Corruption_Detected : BOOL := FALSE;
  Trend_Replay_Race_Detected : BOOL := FALSE;
  Blackbox_Causality_Drift_Detected : BOOL := FALSE;
  Alarm_Order_Reconstruction_Error : BOOL := FALSE;
  Mixed_Authority_Persistence_Detected : BOOL := FALSE;
  Historical_Truth_Epoch : UDINT := 0;
  Historical_Truth_Epoch_Coherent : BOOL := FALSE;
  Historical_Last_Update_MS : UDINT := 0;
  Historical_Lease_Expired : BOOL := TRUE;
  Historical_Last_Error_Code : UDINT := 0;
  Historical_Last_Error_Text : STRING(160) := '';
  Historical_Invalidation_Count : UDINT := 0;
END_VAR

VAR_GLOBAL  (* GVL_RUNTIME_RESOURCE_AUTHORITY *)
  Runtime_Resource_Authority_Valid : BOOL := FALSE;
  Runtime_Resource_Authority_Granted : BOOL := FALSE;
  Runtime_Resource_Quarantine_Active : BOOL := TRUE;
  Deterministic_Cycle_Time_Valid : BOOL := FALSE;
  Task_Jitter_Within_Bounds : BOOL := FALSE;
  Watchdog_Margin_Stable : BOOL := FALSE;
  Runtime_Latency_Stable : BOOL := FALSE;
  Queue_Backlog_Stable : BOOL := FALSE;
  Current_Task_Jitter_US : UDINT := 0;
  Max_Allowed_Task_Jitter_US : UDINT := 10000;
  Current_Runtime_Latency_US : UDINT := 0;
  Max_Allowed_Runtime_Latency_US : UDINT := 20000;
  Current_Fieldbus_Queue_Depth : UDINT := 0;
  Max_Allowed_Fieldbus_Queue_Depth : UDINT := 100;
  Current_Watchdog_Margin_MS : UDINT := 0;
  Minimum_Watchdog_Margin_MS : UDINT := 50;
  Hidden_Jitter_Amplification_Detected : BOOL := FALSE;
  Queue_Induced_Authority_Lag_Detected : BOOL := FALSE;
  Watchdog_Near_Death_Oscillation_Detected : BOOL := FALSE;
  Runtime_Starvation_Race_Detected : BOOL := FALSE;
  Cycle_Collapse_SplitBrain_Detected : BOOL := FALSE;
  Heap_Fragmentation_Critical : BOOL := FALSE;
  Fieldbus_Backlog_Saturation_Detected : BOOL := FALSE;
  Runtime_Resource_Authority_Epoch : UDINT := 0;
  Runtime_Resource_Authority_Epoch_Coherent : BOOL := FALSE;
  Runtime_Resource_Last_Update_MS : UDINT := 0;
  Runtime_Resource_Lease_Expired : BOOL := TRUE;
  Runtime_Resource_Last_Error_Code : UDINT := 0;
  Runtime_Resource_Last_Error_Text : STRING(160) := '';
  Runtime_Resource_Invalidation_Count : UDINT := 0;
END_VAR

{attribute 'qualified_only'}
VAR_GLOBAL  (* GVL_Water_Runtime_Supervisory_Publication *)
  G_Supervisory_Valid : BOOL;
  G_Last_Update_MS : UDINT;
  G_Any_Leak_Active : BOOL;
  G_Any_Warning_Active : BOOL;
  G_Any_Degraded_Mapping : BOOL;
  G_Selective_Isolation_Available : BOOL;
  G_Global_Fallback_Active : BOOL;
  G_Active_Global_Close_Path : BOOL;
  G_Active_Safety_Latch : BOOL;
  G_Affected_Hydraulic_Zone : UINT;
  G_Affected_Valve_Group : UINT;
  G_Status_Code : UINT;
  G_Status_Text : STRING(128);
END_VAR

VAR_GLOBAL  (* GVL_RUNTIME_SUSTAINABILITY_FABRIC *)
  Runtime_Sustainability_Valid : BOOL := FALSE;
  Runtime_Sustainability_Granted : BOOL := FALSE;
  Runtime_Sustainability_Quarantine_Active : BOOL := TRUE;
  Deterministic_Cycle_Budget_Stable : BOOL := FALSE;
  Runtime_Queue_Load_Stable : BOOL := FALSE;
  Memory_Fragmentation_Stable : BOOL := FALSE;
  Watchdog_Jitter_Stable : BOOL := FALSE;
  HA_Synchronization_Load_Stable : BOOL := FALSE;
  Historical_Persistence_Load_Stable : BOOL := FALSE;
  Snapshot_Publication_Stable : BOOL := FALSE;
  Distributed_Runtime_Load_Coherent : BOOL := FALSE;
  Runtime_Evolution_Sustainable : BOOL := FALSE;
  Memory_Fragmentation_Drift_Detected : BOOL := FALSE;
  Queue_Saturation_Detected : BOOL := FALSE;
  Historical_Persistence_Amplification_Detected : BOOL := FALSE;
  Watchdog_Jitter_Escalation_Detected : BOOL := FALSE;
  HASynchronization_Overload_Detected : BOOL := FALSE;
  Deterministic_Cycle_Erosion_Detected : BOOL := FALSE;
  Runtime_Sustainability_Epoch : UDINT := 0;
  Runtime_Sustainability_Epoch_Coherent : BOOL := FALSE;
  Runtime_Sustainability_Last_Update_MS : UDINT := 0;
  Runtime_Sustainability_Lease_Expired : BOOL := TRUE;
  Runtime_Sustainability_Last_Error_Code : UDINT := 0;
  Runtime_Sustainability_Last_Error_Text : STRING(160) := '';
  Runtime_Sustainability_Invalidation_Count : UDINT := 0;
END_VAR

VAR_GLOBAL  (* GVL_SEMANTIC_PROGRESS *)
  Semantic_Progress_Epoch : ULINT := 0;
  Semantic_Continuity_Epoch : ULINT := 0;
  Semantic_Forward_Progress_Valid : BOOL := FALSE;
  Semantic_Execution_Continuity_OK : BOOL := FALSE;
  Semantic_Execution_Counter : ULINT := 0;
  Semantic_Last_Execution_Counter : ULINT := 0;
  Semantic_Progress_Last_Update_MS : UDINT := 0;
  Semantic_Progress_Timeout_MS : UDINT := 10000;
  Semantic_Stagnation_Detected : BOOL := FALSE;
  Semantic_Replay_Suspected : BOOL := FALSE;
  Semantic_Livelock_Suspected : BOOL := FALSE;
  Semantic_Deadlock_Suspected : BOOL := FALSE;
  Semantic_Progress_Lease_Active : BOOL := FALSE;
  Semantic_Progress_Lease_Expired : BOOL := FALSE;
  Semantic_Progress_Quarantine_Active : BOOL := FALSE;
  Semantic_Runtime_Barrier_Epoch : ULINT := 0;
  Semantic_Runtime_Snapshot_Epoch : ULINT := 0;
  Semantic_Distributed_Commit_Epoch : ULINT := 0;
  Semantic_Output_Publication_Epoch : ULINT := 0;
  Semantic_Last_Runtime_Barrier_Epoch : ULINT := 0;
  Semantic_Last_Runtime_Snapshot_Epoch : ULINT := 0;
  Semantic_Last_Distributed_Commit_Epoch : ULINT := 0;
  Semantic_Last_Output_Publication_Epoch : ULINT := 0;
  Semantic_Runtime_Barrier_Evidence_OK : BOOL := FALSE;
  Semantic_Runtime_Snapshot_Evidence_OK : BOOL := FALSE;
  Semantic_Distributed_Commit_Evidence_OK : BOOL := FALSE;
  Semantic_Output_Publication_Evidence_OK : BOOL := FALSE;
  Semantic_Phase_Evidence_OK : BOOL := FALSE;
  Semantic_Phase_Stall_Detected : BOOL := FALSE;
  Semantic_Output_Stall_Detected : BOOL := FALSE;
  Semantic_Last_Error_Code : UDINT := 0;
  Semantic_Last_Error_Text : STRING(160) := '';
  Semantic_Invalidation_Count : UDINT := 0;
END_VAR

{attribute 'qualified_only'}
VAR_GLOBAL  (* GVL_Predictive_Diagnostics *)
  G_Diagnostics_State : ARRAY[1..64] OF ST_Predictive_Diagnostics_State;
END_VAR

VAR_GLOBAL  (* GVL_ACTUATION_AUTHORITY *)
  Actuation_Authority_Valid : BOOL := FALSE;
  Actuation_Authority_Granted : BOOL := FALSE;
  Actuation_Quarantine_Active : BOOL := TRUE;
  Actuation_Command_Epoch : UDINT := 0;
  Field_ACK_Epoch : UDINT := 0;
  Actuation_Authority_Epoch : UDINT := 0;
  Field_Device_ACK_Valid : BOOL := FALSE;
  Actuator_Transition_Observed : BOOL := FALSE;
  Physical_Convergence_Confirmed : BOOL := FALSE;
  Stable_Physical_Convergence : BOOL := FALSE;
  Current_Signature_Confirmed : BOOL := FALSE;
  Flow_Response_Confirmed : BOOL := FALSE;
  Pressure_Response_Confirmed : BOOL := FALSE;
  Motion_Response_Confirmed : BOOL := FALSE;
  Stale_Field_ACK_Detected : BOOL := FALSE;
  Write_Without_Confirm_Detected : BOOL := FALSE;
  Relay_Weld_Suspected : BOOL := FALSE;
  Actuator_Stall_Detected : BOOL := FALSE;
  Partial_Actuation_Detected : BOOL := FALSE;
  Command_Actuation_Skew_Detected : BOOL := FALSE;
  ACK_Replay_Suspected : BOOL := FALSE;
  Actuation_Last_Update_MS : UDINT := 0;
  Actuation_Lease_Expired : BOOL := TRUE;
  Actuation_Last_Error_Code : UDINT := 0;
  Actuation_Last_Error_Text : STRING(160) := '';
  Actuation_Invalidation_Count : UDINT := 0;
END_VAR

VAR_GLOBAL  (* GVL_GOVERNANCE_LIVENESS_INTEGRITY_FABRIC *)
  Governance_Liveness_Integrity_Valid : BOOL := FALSE;
  Governance_Liveness_Integrity_Granted : BOOL := FALSE;
  Governance_Liveness_Integrity_Quarantine_Active : BOOL := TRUE;
  Governance_Execution_Liveness_Stable : BOOL := FALSE;
  Integrity_Governor_Scheduling_Canonical : BOOL := FALSE;
  CrossGovernor_Execution_Continuity_Valid : BOOL := FALSE;
  Deterministic_Validation_Cycle_Integrity : BOOL := FALSE;
  Governance_Runtime_Liveness_Coherent : BOOL := FALSE;
  Validation_Cycle_Timing_Monotonic : BOOL := FALSE;
  Distributed_Governor_Execution_Aligned : BOOL := FALSE;
  Runtime_Integrity_Causality_Grounded : BOOL := FALSE;
  Governance_Execution_Budget_Stable : BOOL := FALSE;
  Integrity_Governor_Starvation_Detected : BOOL := FALSE;
  Validation_Cycle_Skip_Detected : BOOL := FALSE;
  CrossGovernor_Execution_Jitter_Fork : BOOL := FALSE;
  Selective_Governance_Degradation_Detected : BOOL := FALSE;
  Runtime_Governor_Execution_Stall_Detected : BOOL := FALSE;
  Distributed_Liveness_Reality_Fork_Detected : BOOL := FALSE;
  Governance_Liveness_Integrity_Epoch : UDINT := 0;
  Governance_Liveness_Integrity_Epoch_Coherent : BOOL := FALSE;
  Governance_Liveness_Integrity_Last_Update_MS : UDINT := 0;
  Governance_Liveness_Integrity_Lease_Expired : BOOL := TRUE;
  Governance_Liveness_Integrity_Last_Error_Code : UDINT := 0;
  Governance_Liveness_Integrity_Last_Error_Text : STRING(160) := '';
  Governance_Liveness_Integrity_Invalidation_Count : UDINT := 0;
END_VAR

VAR_GLOBAL  (* GVL_BEHAVIOR_ADAPT *)
  G_Behavior_Weight_Comfort : REAL := 1.0;
  G_Behavior_Weight_Night : REAL := 1.0;
  G_Behavior_Weight_Preheat : REAL := 1.0;
  G_Behavior_Weight_VentBoost : REAL := 1.0;
  G_Behavior_Weight_AccessSecure : REAL := 1.0;
  G_Scenario_Stats : ARRAY[0..10] OF ST_Scenario_Stats;
  G_VentBoost_Zone_Adapt : ARRAY[1..GVL_CONSTANTS.C_MAX_ZONES] OF ST_Zone_Adapt_State;
  G_Adapt_Profile : E_Adapt_Profile := ADAPT_PROFILE_BALANCED;
  G_Adapt_Enabled : BOOL := TRUE;
  G_Adapt_Learning_Rate : REAL := 0.05;
  G_Adapt_Update_Threshold : INT := 5;
  G_Adapt_Min_Confidence : REAL := 0.30;
  G_Adapt_Default_Zone_Weight : REAL := 1.0;
  G_Confidence_Learning_Rate : REAL := 0.05;
  G_Decay_Factor : REAL := 0.995;
  G_Prev_Humidity : ARRAY[1..GVL_CONSTANTS.C_MAX_ZONES] OF REAL;
  G_Prev_Valid : ARRAY[1..GVL_CONSTANTS.C_MAX_ZONES] OF BOOL;
END_VAR

VAR_GLOBAL  (* GVL_SEMANTIC_DRIFT_OBSERVABILITY_FABRIC *)
  Semantic_Drift_Observability_Active : BOOL := TRUE;
  Semantic_Continuity_Observed : BOOL := FALSE;
  Semantic_Projection_Consistency_Observed : BOOL := FALSE;
  Distributed_Semantic_Alignment_Observed : BOOL := FALSE;
  Semantic_Drift_ReadOnly_Mode : BOOL := TRUE;
  Semantic_Drift_NoExecutionMutation : BOOL := TRUE;
  Semantic_Drift_Observed : BOOL := FALSE;
  Semantic_Lineage_Drift_Observed : BOOL := FALSE;
  Semantic_Projection_Decay_Observed : BOOL := FALSE;
  Semantic_Drift_Observation_Epoch : UDINT := 0;
END_VAR

VAR_GLOBAL  (* GVL_COMMAND_VERIFY *)
  Command_Mismatch_Count : INT := 0;
  Command_Match_OK : BOOL := TRUE;
  Command_Mismatch_Active : BOOL := FALSE;
  Runtime_Sanity_OK : BOOL := TRUE;
  Runtime_Sanity_Error_Count : UDINT := 0;
  Runtime_Last_Error_Code : UDINT := 0;
  Runtime_Last_Error_Time_MS : UDINT := 0;
  Runtime_Last_Error_Text : STRING(160) := '';
  PreOutput_Barrier_OK : BOOL := TRUE;
  PreOutput_Block_IO : BOOL := FALSE;
  PreOutput_Physical_Causality_Valid : BOOL := FALSE;
  PreOutput_Block_Count : UDINT := 0;
  PreOutput_Last_Error_Code : UDINT := 0;
  PreOutput_Last_Error_Time_MS : UDINT := 0;
  PreOutput_Last_Error_Text : STRING(160) := '';
END_VAR

VAR_GLOBAL  (* GVL_RESIDUAL_ENERGY_STATE_FABRIC *)
  Residual_Energy_State_Valid : BOOL := FALSE;
  Residual_Energy_Bounded : BOOL := FALSE;
  Residual_Actuation_Energy_Safe : BOOL := FALSE;
  Thermal_Energy_Dissipation_Stable : BOOL := FALSE;
  Residual_Energy_Causality_Valid : BOOL := FALSE;
  Distributed_Residual_Energy_Consensus : BOOL := FALSE;
  Latent_Unsafe_Actuation_Detected : BOOL := FALSE;
  Residual_Energy_Persistence_Detected : BOOL := FALSE;
  Unsafe_Thermal_Energy_Retention : BOOL := FALSE;
  Residual_Energy_Epoch : UDINT := 0;
END_VAR

{attribute 'qualified_only'}
VAR_GLOBAL  (* GVL_Cluster_Runtime_FSM *)
  G_State_Startup : BOOL;
  G_State_Discovery : BOOL;
  G_State_Synchronization : BOOL;
  G_State_Operational : BOOL;
  G_State_Degraded : BOOL;
  G_State_Observer_Only : BOOL;
  G_State_Recovery_Lock : BOOL;
  G_State_Quarantine : BOOL;
  G_Runtime_Valid : BOOL;
  G_Last_Update_MS : UDINT;
  G_Status_Code : UINT;
  G_Status_Text : STRING(160);
END_VAR

VAR_GLOBAL  (* GVL_AUTHORITY_PROVENANCE_FABRIC *)
  Authority_Provenance_Valid : BOOL := FALSE;
  Authority_Provenance_Granted : BOOL := FALSE;
  Authority_Provenance_Quarantine_Active : BOOL := TRUE;
  Bootstrap_Authority_Authentic : BOOL := FALSE;
  Commissioning_Lineage_Traceable : BOOL := FALSE;
  Trust_Seed_Integrity_Valid : BOOL := FALSE;
  Root_Authority_Attribution_Coherent : BOOL := FALSE;
  Provenance_Causality_Grounded : BOOL := FALSE;
  Historical_Origin_Lineage_Valid : BOOL := FALSE;
  Distributed_Trust_Chain_Coherent : BOOL := FALSE;
  Authority_Origin_Continuity_Stable : BOOL := FALSE;
  Root_Identity_Cryptographic_Validity : BOOL := FALSE;
  Bootstrap_Identity_Corruption_Detected : BOOL := FALSE;
  Forged_Authority_Root_Detected : BOOL := FALSE;
  Commissioning_Provenance_Gap_Detected : BOOL := FALSE;
  Trust_Seed_Impersonation_Detected : BOOL := FALSE;
  Origin_Authenticity_Erosion_Detected : BOOL := FALSE;
  Root_Lineage_Tampering_Detected : BOOL := FALSE;
  Authority_Provenance_Epoch : UDINT := 0;
  Authority_Provenance_Epoch_Coherent : BOOL := FALSE;
  Authority_Provenance_Last_Update_MS : UDINT := 0;
  Authority_Provenance_Lease_Expired : BOOL := TRUE;
  Authority_Provenance_Last_Error_Code : UDINT := 0;
  Authority_Provenance_Last_Error_Text : STRING(160) := '';
  Authority_Provenance_Invalidation_Count : UDINT := 0;
END_VAR

{attribute 'qualified_only'}
VAR_GLOBAL  (* GVL_Water_Valve_Runtime *)
  G_Valve_Runtime_State : ARRAY[1..64] OF ST_Water_Valve_Runtime_State;
  G_Any_Valve_Degraded : BOOL;
  G_Any_Confirmation_Unknown : BOOL;
  G_Any_Unsafe_Reopen_Denied : BOOL;
  G_Runtime_Valid : BOOL;
  G_Last_Update_MS : UDINT;
  G_Status_Code : UINT;
  G_Status_Text : STRING(128);
END_VAR

{attribute 'qualified_only'}
VAR_GLOBAL  (* GVL_OPENTHERM_ADAPTER *)
  G_Command : ARRAY[1..GVL_CONSTANTS.C_MAX_BOILERS] OF ST_OpenTherm_Command;
  G_Status : ARRAY[1..GVL_CONSTANTS.C_MAX_BOILERS] OF ST_OpenTherm_Status;
  G_Wire_Image : ARRAY[1..GVL_CONSTANTS.C_MAX_BOILERS] OF ST_OpenTherm_Wire_Image;
  G_Transport_Online : BOOL := FALSE;
  G_Transport_Error : BOOL := FALSE;
  G_Last_Transport_Update_MS : UDINT := 0;
END_VAR

{attribute 'qualified_only'}
VAR_GLOBAL  (* GVL_ALARM *)
  G_Security_Armed : BOOL := FALSE;  (* Флаг: Система безопасности активирована *)
  G_Security_Siren : BOOL := FALSE;
  G_Global_Siren : BOOL := FALSE;  (* Глобальный флаг сирены от Alarm Manager *)
  G_Global_Critical : BOOL := FALSE;
  G_Global_Warning : BOOL := FALSE;
  G_Active_Alarm_Count : INT := 0;
  G_Unacked_Alarm_Count : INT := 0;
  G_Alarm_List : ARRAY[1..GVL_CONSTANTS.C_MAX_ALARMS] OF ST_Alarm_Record;
  G_Gas_Alarm_Active : BOOL := FALSE;  (* Флаг: Обнаружена критическая концентрация газа *)
  G_Gas_Fire_Siren : BOOL := FALSE;
  G_Fire_Alarm_Active : BOOL := FALSE;  (* Флаг: Сработали пожарные датчики *)
  G_Flood_Alarm_Active : BOOL := FALSE;  (* Флаг: Обнаружена протечка воды *)
  G_Security_Alarm : BOOL := FALSE;  (* Флаг: Тревога системы безопасности *)
END_VAR

VAR_GLOBAL  (* GVL_EXPLAINABILITY *)
  G_Last_Global_Reason_Code : E_System_Reason_Code := REASON_NONE;
  G_Last_Global_Reason_Text : STRING(255) := 'No active reason';
  G_Last_Safety_Mode : E_Safety_Mode := NORMAL;
  G_Last_Recovery_Phase : E_Recovery_Phase := IDLE;
  G_Last_Command_Source : STRING(80) := '';
  G_Last_Domain_Affected : STRING(80) := '';
  G_Last_Output_Affected : STRING(80) := '';
  G_Last_Update_MS : UDINT := 0;
  G_Behavior_Why_Active : STRING(255) := '';
  G_Heating_Why_Blocked : STRING(255) := '';
  G_Vent_Why_Stopped : STRING(255) := '';
  G_Water_Why_Closed : STRING(255) := '';
  G_Access_Why_Opened : STRING(255) := '';
  G_Reason_Chain_Safety : STRING(80) := 'NORMAL';
  G_Reason_Chain_Behavior : STRING(120) := 'No behavior scenario active';
  G_Reason_Chain_Command : STRING(120) := 'Command OK';
  G_Reason_Chain_Output : STRING(120) := 'Outputs projected';
  G_Reason_Chain_Full : STRING(255) := 'NORMAL -> No behavior scenario active -> Command OK -> Outputs projected';
END_VAR

{attribute 'qualified_only'}
VAR_GLOBAL  (* GVL_Heating_Runtime_Explainability *)
  G_Runtime_Phase_Event : ST_Heating_Runtime_Phase_Event;
  G_Runtime_Anomaly : ST_Heating_Runtime_Anomaly;
  G_Runtime_Blackbox_Event : ST_Heating_Runtime_Blackbox_Event;
  G_Runtime_Blackbox_Timeline : ST_Heating_Runtime_Blackbox_Timeline;
  G_Runtime_Event_Buffer : ST_Heating_Runtime_Event_Buffer;
  G_Runtime_Adaptive_Intelligence : ST_Heating_Runtime_Adaptive_Intelligence;
  G_Runtime_Causality_Graph : ST_Heating_Runtime_Causality_Graph;
  G_Runtime_Integration_Bridge : ST_Heating_Runtime_Integration_Bridge;
  G_Runtime_Predictive_State : ST_Heating_Runtime_Predictive_State;
  G_Runtime_Execution_Timeline : ST_Heating_Runtime_Execution_Timeline;
  G_Runtime_Phase_Transition : ST_Heating_Runtime_Phase_Transition;
  G_Runtime_Explainability_Publication_Valid : BOOL := FALSE;
  G_Runtime_Explainability_Status_Code : UINT := 0;
  G_Runtime_Explainability_Status_Text : STRING(128) := 'Heating runtime explainability inactive';
END_VAR

VAR_GLOBAL  (* GVL_HISTORICAL_ORDERING_INTEGRITY_FABRIC *)
  Historical_Ordering_Integrity_Valid : BOOL := FALSE;
  Historical_Ordering_Integrity_Granted : BOOL := FALSE;
  Historical_Ordering_Integrity_Granted_Proof : BOOL := FALSE;
  Historical_Timeline_Canonical : BOOL := FALSE;
  Forensic_Ordering_Coherent : BOOL := FALSE;
  Historical_Causality_Grounded : BOOL := FALSE;
  Distributed_Historical_Consensus_Valid : BOOL := FALSE;
  Historical_Order_Divergence : BOOL := FALSE;
  Unsafe_Historical_Rewrite_Detected : BOOL := FALSE;
  Historical_Causality_Gap_Detected : BOOL := FALSE;
  Historical_Ordering_Epoch : UDINT := 0;
END_VAR

VAR_GLOBAL  (* GVL_SEMANTIC_EXECUTION_CONTROL *)
  Semantic_Execution_Control_Active : BOOL := TRUE;
  Semantic_Execution_Control_ReadOnly : BOOL := TRUE;
  Temporal_Verification_Domain_Active : BOOL := TRUE;
  Authority_Verification_Domain_Active : BOOL := TRUE;
  Physical_Verification_Domain_Active : BOOL := TRUE;
  Runtime_Verification_Domain_Active : BOOL := TRUE;
  Survivability_Verification_Domain_Active : BOOL := TRUE;
  Safety_Execution_Path : E_SEMANTIC_EXECUTION_PATH := FAST_PATH;
  Physical_Verification_Path : E_SEMANTIC_EXECUTION_PATH := FAST_PATH;
  Runtime_Verification_Path : E_SEMANTIC_EXECUTION_PATH := NORMAL_PATH;
  Diagnostics_Execution_Path : E_SEMANTIC_EXECUTION_PATH := DEFERRED_PATH;
  Trend_Analytics_Execution_Path : E_SEMANTIC_EXECUTION_PATH := BACKGROUND_PATH;
  Semantic_Execution_Fragmentation_Risk : BOOL := FALSE;
  Semantic_Cascade_Amplification_Risk : BOOL := FALSE;
  Semantic_Complexity_Ceiling_Reached : BOOL := FALSE;
  Semantic_Chain_Depth_Limit_Reached : BOOL := FALSE;
  Verification_Fanout_Limit_Reached : BOOL := FALSE;
  Observability_Fanout_Limit_Reached : BOOL := FALSE;
  Lifecycle_Transition_Limit_Reached : BOOL := FALSE;
  Autonomous_Complexity_Ceiling_Enforced : BOOL := FALSE;
  Semantic_Scheduler_Active : BOOL := TRUE;
  Semantic_Execution_Control_Epoch : UDINT := 0;
END_VAR

VAR_GLOBAL  (* GVL_FABRIC_LIFECYCLE_REGISTRY *)
  Fabric_Lifecycle_Registry_Active : BOOL := TRUE;
  Fabric_Lifecycle_Registry_ReadOnly : BOOL := TRUE;
  Runtime_Adaptive_Mode : E_RUNTIME_ADAPTIVE_MODE := FULL_SEMANTIC_MODE;
  Safety_Fabric_State : E_FABRIC_LIFECYCLE_STATE := FABRIC_ACTIVE;
  Authority_Fabric_State : E_FABRIC_LIFECYCLE_STATE := FABRIC_ACTIVE;
  Physical_Reality_Fabric_State : E_FABRIC_LIFECYCLE_STATE := FABRIC_ACTIVE;
  Survivability_Fabric_State : E_FABRIC_LIFECYCLE_STATE := FABRIC_ACTIVE;
  Observability_Fabric_State : E_FABRIC_LIFECYCLE_STATE := FABRIC_ACTIVE;
  Analytics_Fabric_State : E_FABRIC_LIFECYCLE_STATE := FABRIC_ACTIVE;
  Controlled_Capability_Shedding_Allowed : BOOL := FALSE;
  NonEssential_Analytics_Shedding_Recommended : BOOL := FALSE;
  Extended_Observability_Shedding_Recommended : BOOL := FALSE;
  Simulation_Suspension_Recommended : BOOL := FALSE;
  Diagnostics_Degradation_Recommended : BOOL := FALSE;
  Safety_Fabric_Protected : BOOL := TRUE;
  Authority_Fabric_Protected : BOOL := TRUE;
  Physical_Reality_Fabric_Protected : BOOL := TRUE;
  Runtime_Barrier_Protected : BOOL := TRUE;
  Gradual_Reactivation_Allowed : BOOL := FALSE;
  Stability_Validated_Reactivation_Required : BOOL := TRUE;
  Fabric_Lifecycle_Registry_Epoch : UDINT := 0;
END_VAR

{attribute 'qualified_only'}
VAR_GLOBAL  (* GVL_Distributed_Authority *)
  G_Authority_State : ST_Distributed_Authority_State;
  G_Master_Controller_Id : UINT;
  G_Backup_Controller_Id : UINT;
  G_Authority_Lease_Start_MS : UDINT;
  G_Authority_Lease_Duration_MS : UDINT := 30000;
END_VAR

{attribute 'qualified_only'}
VAR_GLOBAL  (* GVL_Water_Valve_Feedback *)
  G_Valve_Feedback_State : ARRAY[1..64] OF ST_Water_Valve_Feedback_State;
  G_Any_Degraded : BOOL;
  G_Any_Timeout : BOOL;
  G_Any_Conflict : BOOL;
  G_Runtime_Valid : BOOL;
  G_Last_Update_MS : UDINT;
  G_Status_Code : UINT;
  G_Status_Text : STRING(128);
END_VAR

VAR_GLOBAL  (* GVL_RECOVERY_ORDERING_INTEGRITY_FABRIC *)
  Recovery_Ordering_Integrity_Valid : BOOL := FALSE;
  CrossDomain_Recovery_Ordering_Stable : BOOL := FALSE;
  Recovery_Authority_Sequencing_Canonical : BOOL := FALSE;
  Physical_Reactivation_Topology_Safe : BOOL := FALSE;
  Recovery_Ordering_Causality_Valid : BOOL := FALSE;
  Distributed_Recovery_Ordering_Consensus : BOOL := FALSE;
  Unsafe_Recovery_Reordering_Detected : BOOL := FALSE;
  CrossDomain_Reactivation_Race : BOOL := FALSE;
  Recovery_Topology_Divergence : BOOL := FALSE;
  Residual_Unsafe_Reactivation_Detected : BOOL := FALSE;
  Recovery_Ordering_Epoch : UDINT := 0;
END_VAR

{attribute 'qualified_only'}
VAR_GLOBAL  (* GVL_MODBUS_SCAN *)
  G_Scan_Enable : BOOL := FALSE;
  G_Scan_Active : BOOL := FALSE;
  G_Scan_Done : BOOL := FALSE;
  G_Scan_Error : BOOL := FALSE;
  G_Slave_ID : BYTE := 1;
  G_Start_Register : UINT := 0;
  G_End_Register : UINT := 255;
  G_Current_Register : UINT := 0;
  G_Found_Register : ARRAY[0..255] OF BOOL;
  G_Found_Value : ARRAY[0..255] OF WORD;
  G_Last_Scan_MS : UDINT := 0;
END_VAR

{attribute 'qualified_only'}
VAR_GLOBAL  (* GVL_IO_Binding_Config *)
  G_Flood_Sensor_Binding : ARRAY[1..64] OF ST_IO_Binding_Record;
  G_Water_Valve_Open_FB_Binding : ARRAY[1..64] OF ST_IO_Binding_Record;
  G_Water_Valve_Close_FB_Binding : ARRAY[1..64] OF ST_IO_Binding_Record;
  G_Water_Valve_Output_Binding : ARRAY[1..64] OF ST_IO_Binding_Record;
END_VAR

{attribute 'qualified_only'}
VAR_GLOBAL  (* GVL_MODBUS_MASTER *)
  G_Request : ARRAY[1..16] OF ST_Modbus_Request;
  G_Response : ARRAY[1..16] OF ST_Modbus_Response;
  G_Master_Online : BOOL := FALSE;
  G_Master_Error : BOOL := FALSE;
  G_Last_Transaction_MS : UDINT := 0;
  G_Active : BOOL := FALSE;
  G_Active_Index : INT := 0;
  G_Active_Sequence : UDINT := 0;
  G_Active_Start_MS : UDINT := 0;
  G_Active_Retry_Count : INT := 0;
  G_Total_Transactions : UDINT := 0;
  G_Total_Errors : UDINT := 0;
  G_Total_Timeouts : UDINT := 0;
END_VAR

VAR_GLOBAL  (* GVL_SEMANTIC_FEDERATION_FABRIC *)
  Semantic_Federation_Valid : BOOL := FALSE;
  Semantic_Federation_Granted : BOOL := FALSE;
  Semantic_Federation_Quarantine_Active : BOOL := TRUE;
  External_SCADA_Semantics_Coherent : BOOL := FALSE;
  Cloud_Authority_Projection_Aligned : BOOL := FALSE;
  MQTT_Semantic_State_Fresh : BOOL := FALSE;
  ThirdParty_Integration_Trust_Valid : BOOL := FALSE;
  Federated_Observability_Coherent : BOOL := FALSE;
  Exported_Authority_State_Coherent : BOOL := FALSE;
  Federation_Projection_Temporal_Stable : BOOL := FALSE;
  External_Runtime_Interpretation_Aligned : BOOL := FALSE;
  Federated_Trust_Boundary_Stable : BOOL := FALSE;
  External_Semantic_Lag_Detected : BOOL := FALSE;
  SCADA_Projection_Skew_Detected : BOOL := FALSE;
  Cloud_Authority_Desynchronization_Detected : BOOL := FALSE;
  ThirdParty_Semantic_Drift_Detected : BOOL := FALSE;
  Integration_Trust_Divergence_Detected : BOOL := FALSE;
  Federated_Authority_Inconsistency_Detected : BOOL := FALSE;
  Semantic_Federation_Epoch : UDINT := 0;
  Semantic_Federation_Epoch_Coherent : BOOL := FALSE;
  Semantic_Federation_Last_Update_MS : UDINT := 0;
  Semantic_Federation_Lease_Expired : BOOL := TRUE;
  Semantic_Federation_Last_Error_Code : UDINT := 0;
  Semantic_Federation_Last_Error_Text : STRING(160) := '';
  Semantic_Federation_Invalidation_Count : UDINT := 0;
END_VAR

VAR_GLOBAL  (* GVL_Heating_Runtime_Observation *)
  G_Runtime_Observer_Lifecycle_State : E_Runtime_Observer_Lifecycle_State := E_Runtime_Observer_Lifecycle_State.ROS_INACTIVE;
  G_Runtime_Observer_Lifecycle_Code : UINT := 0;
  G_Runtime_Observer_Lifecycle_Text : STRING(128) := 'Heating runtime observer inactive';
  G_Runtime_Observer_Commissioning_Required : BOOL := TRUE;
  G_Runtime_Observer_Commissioning_Active : BOOL := FALSE;
  G_Runtime_Observer_Commissioning_Complete : BOOL := FALSE;
  G_Runtime_Observation : ST_Heating_Runtime_Observation;
  G_Runtime_Observation_Publication_Valid : BOOL := FALSE;
  G_Runtime_Observation_Stabilization_Complete : BOOL := FALSE;
  G_Runtime_Observation_Operational : BOOL := FALSE;
  G_Runtime_Observation_Valid : BOOL := FALSE;
  G_Runtime_Observer_Ready : BOOL := FALSE;
  G_Runtime_Observer_Fault : BOOL := FALSE;
  G_Runtime_Observation_Status_Code : UINT := 0;
  G_Runtime_Observation_Status_Text : STRING(128) := 'Heating runtime observation inactive';
END_VAR

VAR_GLOBAL  (* GVL_RUNTIME_ASSUMPTION_INTEGRITY_FABRIC *)
  Runtime_Assumption_Integrity_Active : BOOL := TRUE;
  Runtime_Assumption_Integrity_Observed : BOOL := FALSE;
  Runtime_Assumption_Lineage_Coherent : BOOL := FALSE;
  Runtime_Assumption_Stability_Observed : BOOL := FALSE;
  Runtime_Assumption_ReadOnly_Mode : BOOL := TRUE;
  Runtime_Assumption_NoAuthorityMutation : BOOL := TRUE;
  Runtime_Assumption_Decay_Observed : BOOL := FALSE;
  Runtime_Assumption_Violation_Observed : BOOL := FALSE;
  Runtime_Assumption_Drift_Observed : BOOL := FALSE;
  Runtime_Assumption_Integrity_Epoch : UDINT := 0;
END_VAR

VAR_GLOBAL  (* GVL_SENSOR_CONSENSUS *)
  Sensor_Consensus_Valid : BOOL := FALSE;
  Sensor_Consensus_Quarantine_Active : BOOL := TRUE;
  Sensor_Consensus_Lease_Expired : BOOL := TRUE;
  Physics_Invariants_Satisfied : BOOL := FALSE;
  Cross_Sensor_Correlation_Valid : BOOL := FALSE;
  Telemetry_Plausibility_Valid : BOOL := FALSE;
  Sensor_Drift_Detected : BOOL := FALSE;
  Sensor_Partition_Detected : BOOL := FALSE;
  Sensor_Hallucination_Suspected : BOOL := FALSE;
  Cross_Sensor_Divergence_Detected : BOOL := FALSE;
  Flow_Response_Valid : BOOL := FALSE;
  Pressure_Response_Valid : BOOL := FALSE;
  Airflow_Response_Valid : BOOL := FALSE;
  Current_Signature_Valid : BOOL := FALSE;
  Sensor_Consensus_Epoch : UDINT := 0;
  Last_Consensus_Update_MS : UDINT := 0;
  Sensor_Consensus_Freshness_Valid : BOOL := FALSE;
  Sensor_Oscillation_Detected : BOOL := FALSE;
  Sensor_Stuck_State_Detected : BOOL := FALSE;
  Sensor_Replay_Suspected : BOOL := FALSE;
  Sensor_Consensus_Last_Error_Code : UDINT := 0;
  Sensor_Consensus_Last_Error_Text : STRING(160) := '';
  Sensor_Consensus_Invalidation_Count : UDINT := 0;
END_VAR

{attribute 'qualified_only'}
VAR_GLOBAL  (* GVL_Runtime_Bus *)
  G_TX_Frames : ARRAY[1..128] OF ST_Runtime_Bus_Frame;
  G_RX_Frames : ARRAY[1..128] OF ST_Runtime_Bus_Frame;
END_VAR

{attribute 'qualified_only'}
VAR_GLOBAL  (* GVL_Runtime_Sessions *)
  G_Local_Session : ST_Runtime_Node_Session;
  G_Remote_Sessions : ARRAY[1..16] OF ST_Runtime_Node_Session;
END_VAR

{attribute 'qualified_only'}
VAR_GLOBAL  (* GVL_Cluster_Safety_Barrier *)
  G_Runtime_Valid : BOOL;
  G_Last_Update_MS : UDINT;
  G_Cluster_Execution_Blocked : BOOL;
  G_Authority_Downgraded : BOOL;
  G_Orchestration_Restricted : BOOL;
  G_Remote_Authority_Degraded : BOOL;
  G_Runtime_Bus_Degraded : BOOL;
  G_Projection_Ownership_Invalid : BOOL;
  G_Recovery_Lock_Active : BOOL;
  G_Deployment_Invalid : BOOL;
  G_Status_Code : UINT;
  G_Status_Text : STRING(160);
END_VAR

